IF st_config_achse.b_config_fertig THEN
	(* Fehlermeldungen und Betriebsmeldungen ab dem Startindex in die globalen Meldungsarrays schreiben *)
	garr_stoermeldungen[st_config_achse.i16_meld_startindex + 0] := st_sm.b_achse_nicht_bb;
	garr_stoermeldungen[st_config_achse.i16_meld_startindex + 1] := st_sm.b_achse_nicht_referenziert;
	garr_stoermeldungen[st_config_achse.i16_meld_startindex + 2] := st_sm.b_keine_verfahrfreigabe;
	garr_stoermeldungen[st_config_achse.i16_meld_startindex + 3] := st_sm.b_achse_nicht_auf_startpos;
	garr_stoermeldungen[st_config_achse.i16_meld_startindex + 4] := st_sm.b_ende_skalierungs_nocke;
	garr_stoermeldungen[st_config_achse.i16_meld_startindex + 5] := st_sm.b_ende_camming_nocke;
	garr_stoermeldungen[st_config_achse.i16_meld_startindex + 6] := st_sm.b_skalierung_noch_aktiv;
	garr_stoermeldungen[st_config_achse.i16_meld_startindex + 7] := FALSE;
	garr_stoermeldungen[st_config_achse.i16_meld_startindex + 8] := FALSE;
	garr_stoermeldungen[st_config_achse.i16_meld_startindex + 9] := sm_fehler_raster_oder_zaehne;
	garr_stoermeldungen[st_config_achse.i16_meld_startindex + 10] := FALSE;
	garr_stoermeldungen[st_config_achse.i16_meld_startindex + 11] := FALSE;
	garr_stoermeldungen[st_config_achse.i16_meld_startindex + 12] := sm_fehler_achse_lueften;
	garr_stoermeldungen[st_config_achse.i16_meld_startindex + 13] := sm_keine_busverbindung;
	garr_stoermeldungen[st_config_achse.i16_meld_startindex + 14] := sm_fehler_bestueckanzahl;
	garr_stoermeldungen[st_config_achse.i16_meld_startindex + 15] := sm_fehler_nach_bandwechsel;
	garr_stoermeldungen[st_config_achse.i16_meld_startindex + 16] := st_drive_cmd.meldungen.sm_write_soe_parameter;
	garr_stoermeldungen[st_config_achse.i16_meld_startindex + 17] := st_drive_cmd.meldungen.sm_read_soe_parameter;
	garr_stoermeldungen[st_config_achse.i16_meld_startindex + 18] := st_drive_cmd.meldungen.sm_write_nc_parameter;
	garr_stoermeldungen[st_config_achse.i16_meld_startindex + 19] := st_drive_cmd.meldungen.sm_read_nc_parameter;
	garr_stoermeldungen[st_config_achse.i16_meld_startindex + 20] := st_drive_cmd.meldungen.sm_power_enable;
	garr_stoermeldungen[st_config_achse.i16_meld_startindex + 21] := st_drive_cmd.meldungen.sm_power_disable;
	garr_stoermeldungen[st_config_achse.i16_meld_startindex + 22] := st_drive_cmd.meldungen.sm_reset;
	garr_stoermeldungen[st_config_achse.i16_meld_startindex + 23] := st_drive_cmd.meldungen.sm_home;
	garr_stoermeldungen[st_config_achse.i16_meld_startindex + 24] := st_drive_cmd.meldungen.sm_setposition;
	garr_stoermeldungen[st_config_achse.i16_meld_startindex + 25] := st_drive_cmd.meldungen.sm_jog_vorwaerts;
	garr_stoermeldungen[st_config_achse.i16_meld_startindex + 26] := st_drive_cmd.meldungen.sm_jog_rueckwaerts;
	garr_stoermeldungen[st_config_achse.i16_meld_startindex + 27] := st_drive_cmd.meldungen.sm_move_absolute;
	garr_stoermeldungen[st_config_achse.i16_meld_startindex + 28] := st_drive_cmd.meldungen.sm_move_relative;
	garr_stoermeldungen[st_config_achse.i16_meld_startindex + 29] := st_drive_cmd.meldungen.sm_move_velocity;
	garr_stoermeldungen[st_config_achse.i16_meld_startindex + 30] := st_drive_cmd.meldungen.sm_move_modulo;
	garr_stoermeldungen[st_config_achse.i16_meld_startindex + 31] := st_drive_cmd.meldungen.sm_stop_axis;
	garr_stoermeldungen[st_config_achse.i16_meld_startindex + 32] := st_drive_cmd.meldungen.sm_halt_axis;
	garr_stoermeldungen[st_config_achse.i16_meld_startindex + 33] := st_drive_cmd.meldungen.sm_motion_command_timeout;
	garr_stoermeldungen[st_config_achse.i16_meld_startindex + 34] := st_sm.b_achsfehler;
	garr_stoermeldungen[st_config_achse.i16_meld_startindex + 35] := st_sm.b_devicefehler;
	garr_stoermeldungen[st_config_achse.i16_meld_startindex + 36] := st_drive_cmd.meldungen.sm_limit_positiv_erreicht;
	garr_stoermeldungen[st_config_achse.i16_meld_startindex + 37] := st_drive_cmd.meldungen.sm_limit_negativ_erreicht;
	garr_stoermeldungen[st_config_achse.i16_meld_startindex + 38] := st_drive_cmd.meldungen.sm_ec_coe_sdo_write_ex;
	garr_stoermeldungen[st_config_achse.i16_meld_startindex + 39] := st_drive_cmd.meldungen.sm_ec_coe_sdo_read_ex;
	garr_stoermeldungen[st_config_achse.i16_meld_startindex + 40] := st_drive_cmd_z_achse.meldungen.sm_gear_in_slave;
	garr_stoermeldungen[st_config_achse.i16_meld_startindex + 41] := st_drive_cmd_z_achse.meldungen.sm_gear_out_slave;
	garr_stoermeldungen[st_config_achse.i16_meld_startindex + 42] := st_drive_cmd_z_achse.meldungen.sm_cam_in_slave;
	garr_stoermeldungen[st_config_achse.i16_meld_startindex + 43] := st_drive_cmd_z_achse.meldungen.sm_cam_out_slave;
	garr_stoermeldungen[st_config_achse.i16_meld_startindex + 44] := st_drive_cmd_z_achse.meldungen.sm_cam_scaleing_slave;
	garr_stoermeldungen[st_config_achse.i16_meld_startindex + 45] := st_drive_cmd_z_achse.meldungen.sm_camgear_command_timeout;
	garr_stoermeldungen[st_config_achse.i16_meld_startindex + 46] := st_drive_cmd_z_achse.meldungen.sm_read_motion_funktion_point;
	garr_stoermeldungen[st_config_achse.i16_meld_startindex + 47] := st_drive_cmd_z_achse.meldungen.sm_write_motion_funktion_point;
	garr_stoermeldungen[st_config_achse.i16_meld_startindex + 48] := st_drive_cmd_z_achse.meldungen.sm_read_camtable_slave_dynamics;
	garr_stoermeldungen[st_config_achse.i16_meld_startindex + 49] := st_drive_cmd_z_achse.meldungen.sm_read_camtable_charakteristik;
	garr_stoermeldungen[st_config_achse.i16_meld_startindex + 50] := st_drive_cmd_y_achse.meldungen.sm_gear_in_slave;
	garr_stoermeldungen[st_config_achse.i16_meld_startindex + 51] := st_drive_cmd_y_achse.meldungen.sm_gear_out_slave;
	garr_stoermeldungen[st_config_achse.i16_meld_startindex + 52] := st_drive_cmd_y_achse.meldungen.sm_cam_in_slave;
	garr_stoermeldungen[st_config_achse.i16_meld_startindex + 53] := st_drive_cmd_y_achse.meldungen.sm_cam_out_slave;
	garr_stoermeldungen[st_config_achse.i16_meld_startindex + 54] := st_drive_cmd_y_achse.meldungen.sm_cam_scaleing_slave;
	garr_stoermeldungen[st_config_achse.i16_meld_startindex + 55] := st_drive_cmd_y_achse.meldungen.sm_camgear_command_timeout;
	garr_stoermeldungen[st_config_achse.i16_meld_startindex + 56] := st_drive_cmd_y_achse.meldungen.sm_read_motion_funktion_point;
	garr_stoermeldungen[st_config_achse.i16_meld_startindex + 57] := st_drive_cmd_y_achse.meldungen.sm_write_motion_funktion_point;
	garr_stoermeldungen[st_config_achse.i16_meld_startindex + 58] := st_drive_cmd_y_achse.meldungen.sm_read_camtable_slave_dynamics;
	garr_stoermeldungen[st_config_achse.i16_meld_startindex + 59] := st_drive_cmd_y_achse.meldungen.sm_read_camtable_charakteristik;
	garr_stoermeldungen[st_config_achse.i16_meld_startindex + 60] := st_drive_cmd_b_achse.meldungen.sm_gear_in_slave;
	garr_stoermeldungen[st_config_achse.i16_meld_startindex + 61] := st_drive_cmd_b_achse.meldungen.sm_gear_out_slave;
	garr_stoermeldungen[st_config_achse.i16_meld_startindex + 62] := st_drive_cmd_b_achse.meldungen.sm_cam_in_slave;
	garr_stoermeldungen[st_config_achse.i16_meld_startindex + 63] := st_drive_cmd_b_achse.meldungen.sm_cam_out_slave;
	garr_stoermeldungen[st_config_achse.i16_meld_startindex + 64] := st_drive_cmd_b_achse.meldungen.sm_cam_scaleing_slave;
	garr_stoermeldungen[st_config_achse.i16_meld_startindex + 65] := st_drive_cmd_b_achse.meldungen.sm_camgear_command_timeout;
	garr_stoermeldungen[st_config_achse.i16_meld_startindex + 66] := st_drive_cmd_b_achse.meldungen.sm_read_motion_funktion_point;
	garr_stoermeldungen[st_config_achse.i16_meld_startindex + 67] := st_drive_cmd_b_achse.meldungen.sm_write_motion_funktion_point;
	garr_stoermeldungen[st_config_achse.i16_meld_startindex + 68] := st_drive_cmd_b_achse.meldungen.sm_read_camtable_slave_dynamics;
	garr_stoermeldungen[st_config_achse.i16_meld_startindex + 69] := st_drive_cmd_b_achse.meldungen.sm_read_camtable_charakteristik;
	garr_stoermeldungen[st_config_achse.i16_meld_startindex + 70] :=  sm_fehler_positionierung_z;
	garr_stoermeldungen[st_config_achse.i16_meld_startindex + 71] :=  sm_fehler_positionierung_y;
	garr_stoermeldungen[st_config_achse.i16_meld_startindex + 72] :=  sm_fehler_bestueckschieberanzahl;
	garr_stoermeldungen[st_config_achse.i16_meld_startindex + 73] :=  sm_fehler_bestueckposition_z;
	garr_stoermeldungen[st_config_achse.i16_meld_startindex + 74] :=  sm_fehler_bestueckposition_y;
	garr_stoermeldungen[st_config_achse.i16_meld_startindex + 75] :=  sm_fehler_positionierung_bestueckachse;
	garr_stoermeldungen[st_config_achse.i16_meld_startindex + 76] :=  st_drive_cmd_bestueckachse.meldungen.sm_gear_in_slave;
	garr_stoermeldungen[st_config_achse.i16_meld_startindex + 77] :=  st_drive_cmd_bestueckachse.meldungen.sm_gear_out_slave;
	garr_stoermeldungen[st_config_achse.i16_meld_startindex + 78] :=  st_drive_cmd_bestueckachse.meldungen.sm_cam_in_slave;
	garr_stoermeldungen[st_config_achse.i16_meld_startindex + 79] :=  st_drive_cmd_bestueckachse.meldungen.sm_cam_out_slave;
	garr_stoermeldungen[st_config_achse.i16_meld_startindex + 80] :=  st_drive_cmd_bestueckachse.meldungen.sm_camgear_command_timeout;
	garr_stoermeldungen[st_config_achse.i16_meld_startindex + 81] :=  st_drive_cmd_bestueckachse.meldungen.sm_read_motion_funktion_point;
	garr_stoermeldungen[st_config_achse.i16_meld_startindex + 82] :=  st_drive_cmd_bestueckachse.meldungen.sm_write_motion_funktion_point;
	garr_stoermeldungen[st_config_achse.i16_meld_startindex + 83] :=  st_drive_cmd_bestueckachse.meldungen.sm_read_camtable_slave_dynamics;
	garr_stoermeldungen[st_config_achse.i16_meld_startindex + 84] :=  st_drive_cmd_bestueckachse.meldungen.sm_read_camtable_charakteristik;
	garr_stoermeldungen[st_config_achse.i16_meld_startindex + 85] :=  FALSE;
	garr_stoermeldungen[st_config_achse.i16_meld_startindex + 86] :=  FALSE;
	garr_stoermeldungen[st_config_achse.i16_meld_startindex + 87] :=  FALSE;
	garr_stoermeldungen[st_config_achse.i16_meld_startindex + 88] :=  FALSE;
	garr_stoermeldungen[st_config_achse.i16_meld_startindex + 89] :=  FALSE;
	garr_stoermeldungen[st_config_achse.i16_meld_startindex + 90] :=  FALSE;
	garr_stoermeldungen[st_config_achse.i16_meld_startindex + 91] :=  FALSE;
	garr_stoermeldungen[st_config_achse.i16_meld_startindex + 92] :=  FALSE;
	garr_stoermeldungen[st_config_achse.i16_meld_startindex + 93] :=  FALSE;
	garr_stoermeldungen[st_config_achse.i16_meld_startindex + 94] :=  FALSE;
	garr_stoermeldungen[st_config_achse.i16_meld_startindex + 95] :=  FALSE;
	garr_stoermeldungen[st_config_achse.i16_meld_startindex + 96] :=  FALSE;
	garr_stoermeldungen[st_config_achse.i16_meld_startindex + 97] :=  FALSE;
	garr_stoermeldungen[st_config_achse.i16_meld_startindex + 98] :=  FALSE;
	garr_stoermeldungen[st_config_achse.i16_meld_startindex + 99] :=  FALSE;
	
	garr_betriebsmeldungen[st_config_achse.i16_meld_startindex + 0] := bm_bandende_einzug_links_erreicht;
	garr_betriebsmeldungen[st_config_achse.i16_meld_startindex + 1] := bm_einzug_links_band_entnehmen;
	garr_betriebsmeldungen[st_config_achse.i16_meld_startindex + 2] := bm_einzug_links_band_auf_anschlag;
	garr_betriebsmeldungen[st_config_achse.i16_meld_startindex + 3] := FALSE;
	garr_betriebsmeldungen[st_config_achse.i16_meld_startindex + 4] := FALSE;
	garr_betriebsmeldungen[st_config_achse.i16_meld_startindex + 5] := FALSE;
	garr_betriebsmeldungen[st_config_achse.i16_meld_startindex + 6] := FALSE;
	garr_betriebsmeldungen[st_config_achse.i16_meld_startindex + 7] := FALSE;
	garr_betriebsmeldungen[st_config_achse.i16_meld_startindex + 8] := FALSE;
	garr_betriebsmeldungen[st_config_achse.i16_meld_startindex + 9] := FALSE;
	garr_betriebsmeldungen[st_config_achse.i16_meld_startindex + 10] := bm_bandende_einzug_rechts_erreicht;
	garr_betriebsmeldungen[st_config_achse.i16_meld_startindex + 11] := bm_einzug_rechts_band_entnehmen;
	garr_betriebsmeldungen[st_config_achse.i16_meld_startindex + 12] := bm_einzug_rechts_band_auf_anschlag;
	garr_betriebsmeldungen[st_config_achse.i16_meld_startindex + 13] := FALSE;
	garr_betriebsmeldungen[st_config_achse.i16_meld_startindex + 14] := FALSE;
	garr_betriebsmeldungen[st_config_achse.i16_meld_startindex + 15] := FALSE;
	garr_betriebsmeldungen[st_config_achse.i16_meld_startindex + 16] := FALSE;
	garr_betriebsmeldungen[st_config_achse.i16_meld_startindex + 17] := FALSE;
	garr_betriebsmeldungen[st_config_achse.i16_meld_startindex + 18] := FALSE;
	garr_betriebsmeldungen[st_config_achse.i16_meld_startindex + 19] := FALSE;
	garr_betriebsmeldungen[st_config_achse.i16_meld_startindex + 20] := bm_bandende_beide_einzuege_erreicht;
	garr_betriebsmeldungen[st_config_achse.i16_meld_startindex + 21] := bm_override_kleiner_stufe9;
	garr_betriebsmeldungen[st_config_achse.i16_meld_startindex + 22] := bm_md_offset_z_pos_0_zu_hoch;
	garr_betriebsmeldungen[st_config_achse.i16_meld_startindex + 23] := bm_md_offset_y_pos_0_zu_hoch;
	garr_betriebsmeldungen[st_config_achse.i16_meld_startindex + 24] := FALSE;
	garr_betriebsmeldungen[st_config_achse.i16_meld_startindex + 25] := FALSE;
	garr_betriebsmeldungen[st_config_achse.i16_meld_startindex + 26] := FALSE;
	garr_betriebsmeldungen[st_config_achse.i16_meld_startindex + 27] := FALSE;
	garr_betriebsmeldungen[st_config_achse.i16_meld_startindex + 28] := FALSE;
	garr_betriebsmeldungen[st_config_achse.i16_meld_startindex + 29] := FALSE;
	garr_betriebsmeldungen[st_config_achse.i16_meld_startindex + 30] := FALSE;
	garr_betriebsmeldungen[st_config_achse.i16_meld_startindex + 31] := FALSE;
	garr_betriebsmeldungen[st_config_achse.i16_meld_startindex + 32] := FALSE;
	garr_betriebsmeldungen[st_config_achse.i16_meld_startindex + 33] := FALSE;
	garr_betriebsmeldungen[st_config_achse.i16_meld_startindex + 34] := FALSE;
	garr_betriebsmeldungen[st_config_achse.i16_meld_startindex + 35] := FALSE;
	garr_betriebsmeldungen[st_config_achse.i16_meld_startindex + 36] := FALSE;
	garr_betriebsmeldungen[st_config_achse.i16_meld_startindex + 37] := FALSE;
	garr_betriebsmeldungen[st_config_achse.i16_meld_startindex + 38] := FALSE;
	garr_betriebsmeldungen[st_config_achse.i16_meld_startindex + 39] := FALSE;
	garr_betriebsmeldungen[st_config_achse.i16_meld_startindex + 40] := FALSE;
	garr_betriebsmeldungen[st_config_achse.i16_meld_startindex + 41] := FALSE;
	garr_betriebsmeldungen[st_config_achse.i16_meld_startindex + 42] := FALSE;
	garr_betriebsmeldungen[st_config_achse.i16_meld_startindex + 43] := FALSE;
	garr_betriebsmeldungen[st_config_achse.i16_meld_startindex + 44] := FALSE;
	garr_betriebsmeldungen[st_config_achse.i16_meld_startindex + 45] := FALSE;
	garr_betriebsmeldungen[st_config_achse.i16_meld_startindex + 46] := FALSE;
	garr_betriebsmeldungen[st_config_achse.i16_meld_startindex + 47] := FALSE;
	garr_betriebsmeldungen[st_config_achse.i16_meld_startindex + 48] := FALSE;
	garr_betriebsmeldungen[st_config_achse.i16_meld_startindex + 49] := FALSE;
	garr_betriebsmeldungen[st_config_achse.i16_meld_startindex + 50] := FALSE;
	garr_betriebsmeldungen[st_config_achse.i16_meld_startindex + 51] := FALSE;
	garr_betriebsmeldungen[st_config_achse.i16_meld_startindex + 52] := FALSE;
	garr_betriebsmeldungen[st_config_achse.i16_meld_startindex + 53] := FALSE;
	garr_betriebsmeldungen[st_config_achse.i16_meld_startindex + 54] := FALSE;
	garr_betriebsmeldungen[st_config_achse.i16_meld_startindex + 55] := FALSE;
	garr_betriebsmeldungen[st_config_achse.i16_meld_startindex + 56] := FALSE;
	garr_betriebsmeldungen[st_config_achse.i16_meld_startindex + 57] := FALSE;
	garr_betriebsmeldungen[st_config_achse.i16_meld_startindex + 58] := FALSE;
	garr_betriebsmeldungen[st_config_achse.i16_meld_startindex + 59] := FALSE;
	garr_betriebsmeldungen[st_config_achse.i16_meld_startindex + 60] := FALSE;
	garr_betriebsmeldungen[st_config_achse.i16_meld_startindex + 61] := FALSE;
	garr_betriebsmeldungen[st_config_achse.i16_meld_startindex + 62] := FALSE;
	garr_betriebsmeldungen[st_config_achse.i16_meld_startindex + 63] := FALSE;
	garr_betriebsmeldungen[st_config_achse.i16_meld_startindex + 64] := FALSE;
	garr_betriebsmeldungen[st_config_achse.i16_meld_startindex + 65] := FALSE;
	garr_betriebsmeldungen[st_config_achse.i16_meld_startindex + 66] := FALSE;
	garr_betriebsmeldungen[st_config_achse.i16_meld_startindex + 67] := FALSE;
	garr_betriebsmeldungen[st_config_achse.i16_meld_startindex + 68] := FALSE;
	garr_betriebsmeldungen[st_config_achse.i16_meld_startindex + 69] := FALSE;
	garr_betriebsmeldungen[st_config_achse.i16_meld_startindex + 70] :=  FALSE;
	garr_betriebsmeldungen[st_config_achse.i16_meld_startindex + 71] :=  FALSE;
	garr_betriebsmeldungen[st_config_achse.i16_meld_startindex + 72] :=  FALSE;
	garr_betriebsmeldungen[st_config_achse.i16_meld_startindex + 73] :=  FALSE;
	garr_betriebsmeldungen[st_config_achse.i16_meld_startindex + 74] :=  FALSE;
	garr_betriebsmeldungen[st_config_achse.i16_meld_startindex + 75] :=  FALSE;
	garr_betriebsmeldungen[st_config_achse.i16_meld_startindex + 76] :=  FALSE;
	garr_betriebsmeldungen[st_config_achse.i16_meld_startindex + 77] :=  FALSE;
	garr_betriebsmeldungen[st_config_achse.i16_meld_startindex + 78] :=  FALSE;
	garr_betriebsmeldungen[st_config_achse.i16_meld_startindex + 79] :=  FALSE;
	garr_betriebsmeldungen[st_config_achse.i16_meld_startindex + 80] :=  FALSE;
	garr_betriebsmeldungen[st_config_achse.i16_meld_startindex + 81] :=  FALSE;
	garr_betriebsmeldungen[st_config_achse.i16_meld_startindex + 82] :=  FALSE;
	garr_betriebsmeldungen[st_config_achse.i16_meld_startindex + 83] :=  FALSE;
	garr_betriebsmeldungen[st_config_achse.i16_meld_startindex + 84] :=  FALSE;
	garr_betriebsmeldungen[st_config_achse.i16_meld_startindex + 85] :=  FALSE;
	garr_betriebsmeldungen[st_config_achse.i16_meld_startindex + 86] :=  FALSE;
	garr_betriebsmeldungen[st_config_achse.i16_meld_startindex + 87] :=  FALSE;
	garr_betriebsmeldungen[st_config_achse.i16_meld_startindex + 88] :=  FALSE;
	garr_betriebsmeldungen[st_config_achse.i16_meld_startindex + 89] :=  FALSE;
	garr_betriebsmeldungen[st_config_achse.i16_meld_startindex + 90] :=  FALSE;
	garr_betriebsmeldungen[st_config_achse.i16_meld_startindex + 91] :=  FALSE;
	garr_betriebsmeldungen[st_config_achse.i16_meld_startindex + 92] :=  FALSE;
	garr_betriebsmeldungen[st_config_achse.i16_meld_startindex + 93] :=  FALSE;
	garr_betriebsmeldungen[st_config_achse.i16_meld_startindex + 94] :=  FALSE;
	garr_betriebsmeldungen[st_config_achse.i16_meld_startindex + 95] :=  FALSE;
	garr_betriebsmeldungen[st_config_achse.i16_meld_startindex + 96] :=  FALSE;
	garr_betriebsmeldungen[st_config_achse.i16_meld_startindex + 97] :=  FALSE;
	garr_betriebsmeldungen[st_config_achse.i16_meld_startindex + 98] :=  FALSE;
	garr_betriebsmeldungen[st_config_achse.i16_meld_startindex + 99] :=  FALSE;
END_IF
END_PROGRAM
ACTION subr_ST_B_Achse:
(* Überwachung, wenn falsche Info aus dem Bestückbild kommt *)
(* Fehler, wenn mehr bestückt werden soll als das WKZ Bestückschieber hat *)
IF gst_datensatz.st_bestueckprogramm.i16_b[i16_bestueckposzaehler] > gst_datensatz.st_wkz.i16_anzahl_bestueckschieber THEN
	sm_fehler_bestueckschieberanzahl := TRUE;
	fb_state_entry.i16_next_step := FEHLER;
END_IF
END_ACTION
ACTION subr_ST_Bandeinzugsnocken_aus:
CASE gst_datensatz.st_wkz.i16_typ_bandeinzug OF
	 STANDARD_2FACH_V2:

		(* Bandeinzug: Standard_2fach_V1 *)
		gst_datensatz.st_wkz.nockenschaltwerk_bestueckachse.arr_nocken[NO_BW_BANDFAENGER_LI_EINFAHREN].b_camvalid := FALSE;
		gst_datensatz.st_wkz.nockenschaltwerk_bestueckachse.arr_nocken[NO_BW_BANDFAENGER_LI_AUSFAHREN].b_camvalid := FALSE;
		gst_datensatz.st_wkz.nockenschaltwerk_bestueckachse.arr_nocken[NO_BW_BANDKLEMMEN_LI_EINFAHREN].b_camvalid := FALSE;
		gst_datensatz.st_wkz.nockenschaltwerk_bestueckachse.arr_nocken[NO_BW_BANDKLEMMEN_LI_AUSFAHREN].b_camvalid := FALSE;
		gst_datensatz.st_wkz.nockenschaltwerk_bestueckachse.arr_nocken[NO_UW_BANDFAENGER_LI_EINFAHREN].b_camvalid := FALSE;
		gst_datensatz.st_wkz.nockenschaltwerk_bestueckachse.arr_nocken[NO_UW_BANDFAENGER_LI_AUSFAHREN].b_camvalid := FALSE;
		gst_datensatz.st_wkz.nockenschaltwerk_bestueckachse.arr_nocken[NO_UW_BANDKLEMMEN_LI_EINFAHREN].b_camvalid := FALSE;
		gst_datensatz.st_wkz.nockenschaltwerk_bestueckachse.arr_nocken[NO_UW_BANDKLEMMEN_LI_AUSFAHREN].b_camvalid := FALSE;
		gst_datensatz.st_wkz.nockenschaltwerk_bestueckachse.arr_nocken[NO_BW_BANDFAENGER_RE_EINFAHREN].b_camvalid := FALSE;
		gst_datensatz.st_wkz.nockenschaltwerk_bestueckachse.arr_nocken[NO_BW_BANDFAENGER_RE_AUSFAHREN].b_camvalid := FALSE;
		gst_datensatz.st_wkz.nockenschaltwerk_bestueckachse.arr_nocken[NO_BW_BANDKLEMMEN_RE_EINFAHREN].b_camvalid := FALSE;
		gst_datensatz.st_wkz.nockenschaltwerk_bestueckachse.arr_nocken[NO_BW_BANDKLEMMEN_RE_AUSFAHREN].b_camvalid := FALSE;
		gst_datensatz.st_wkz.nockenschaltwerk_bestueckachse.arr_nocken[NO_UW_BANDFAENGER_RE_EINFAHREN].b_camvalid := FALSE;
		gst_datensatz.st_wkz.nockenschaltwerk_bestueckachse.arr_nocken[NO_UW_BANDFAENGER_RE_AUSFAHREN].b_camvalid := FALSE;
		gst_datensatz.st_wkz.nockenschaltwerk_bestueckachse.arr_nocken[NO_UW_BANDKLEMMEN_RE_EINFAHREN].b_camvalid := FALSE;
		gst_datensatz.st_wkz.nockenschaltwerk_bestueckachse.arr_nocken[NO_UW_BANDKLEMMEN_RE_AUSFAHREN].b_camvalid := FALSE;
		(* Bandeinzug: Standard_2fach_V2 *)
		gst_datensatz.st_wkz.nockenschaltwerk_bestueckachse.arr_nocken[NO_BW_BANDFAENGER_LI_BAEZV2_EINFAHREN].b_camvalid := FALSE;
		gst_datensatz.st_wkz.nockenschaltwerk_bestueckachse.arr_nocken[NO_BW_BANDFAENGER_LI_BAEZV2_AUSFAHREN].b_camvalid := FALSE;
		gst_datensatz.st_wkz.nockenschaltwerk_bestueckachse.arr_nocken[NO_BW_BANDKLEMMEN_LI_BAEZV2_EINFAHREN].b_camvalid := FALSE;
		gst_datensatz.st_wkz.nockenschaltwerk_bestueckachse.arr_nocken[NO_BW_BANDKLEMMEN_LI_BAEZV2_AUSFAHREN].b_camvalid := FALSE;
		gst_datensatz.st_wkz.nockenschaltwerk_bestueckachse.arr_nocken[NO_BW_BANDFAENGER_RE_BAEZV2_EINFAHREN].b_camvalid := FALSE;
		gst_datensatz.st_wkz.nockenschaltwerk_bestueckachse.arr_nocken[NO_BW_BANDFAENGER_RE_BAEZV2_AUSFAHREN].b_camvalid := FALSE;
		gst_datensatz.st_wkz.nockenschaltwerk_bestueckachse.arr_nocken[NO_BW_BANDKLEMMEN_RE_BAEZV2_EINFAHREN].b_camvalid := FALSE;
		gst_datensatz.st_wkz.nockenschaltwerk_bestueckachse.arr_nocken[NO_BW_BANDKLEMMEN_RE_BAEZV2_AUSFAHREN].b_camvalid := FALSE;

		zyl_bandfaenger_li.fb.b_no_gesteuert_im_norm_betrieb := TRUE;
		zyl_bandklemmen_li.fb.b_no_gesteuert_im_norm_betrieb := TRUE;
		zyl_bandfaenger_re.fb.b_no_gesteuert_im_norm_betrieb := TRUE;
		zyl_bandklemmen_re.fb.b_no_gesteuert_im_norm_betrieb := TRUE;

	BANDWECHSLER_V2:
		(* Klemmbandeinzug ohne Sensoren *)
		gst_datensatz.st_wkz.nockenschaltwerk_bestueckachse.arr_nocken[NO_BW_BANDFAENGER_BAWEV2_EINFAHREN].b_camvalid := FALSE;
		gst_datensatz.st_wkz.nockenschaltwerk_bestueckachse.arr_nocken[NO_BW_BANDFAENGER_BAWEV2_AUSFAHREN].b_camvalid := FALSE;
		gst_datensatz.st_wkz.nockenschaltwerk_bestueckachse.arr_nocken[NO_BW_BANDKLEMMEN_BAWEV2_EINFAHREN].b_camvalid := FALSE;
		gst_datensatz.st_wkz.nockenschaltwerk_bestueckachse.arr_nocken[NO_BW_BANDKLEMMEN_BAWEV2_AUSFAHREN].b_camvalid := FALSE;

		gst_datensatz.st_wkz.nockenschaltwerk_bestueckachse.arr_nocken[NO_BW_BANDFAENGER_EINFAHREN].b_camvalid := FALSE;
		gst_datensatz.st_wkz.nockenschaltwerk_bestueckachse.arr_nocken[NO_BW_BANDFAENGER_AUSFAHREN].b_camvalid := FALSE;
		gst_datensatz.st_wkz.nockenschaltwerk_bestueckachse.arr_nocken[NO_BW_BANDKLEMMEN_EINFAHREN].b_camvalid := FALSE;
		gst_datensatz.st_wkz.nockenschaltwerk_bestueckachse.arr_nocken[NO_BW_BANDKLEMMEN_AUSFAHREN].b_camvalid := FALSE;
		gst_datensatz.st_wkz.nockenschaltwerk_bestueckachse.arr_nocken[NO_UW_BANDFAENGER_EINFAHREN].b_camvalid := FALSE;
		gst_datensatz.st_wkz.nockenschaltwerk_bestueckachse.arr_nocken[NO_UW_BANDFAENGER_AUSFAHREN].b_camvalid := FALSE;
		gst_datensatz.st_wkz.nockenschaltwerk_bestueckachse.arr_nocken[NO_UW_BANDKLEMMEN_EINFAHREN].b_camvalid := FALSE;
		gst_datensatz.st_wkz.nockenschaltwerk_bestueckachse.arr_nocken[NO_UW_BANDKLEMMEN_AUSFAHREN].b_camvalid := FALSE;

		gst_datensatz.st_wkz.nockenschaltwerk_bestueckachse.arr_nocken[NO_PNEUMATIKBANDEINZUG_GLS].b_camvalid := FALSE;
		gst_datensatz.st_wkz.nockenschaltwerk_bestueckachse.arr_nocken[NO_UW_BESTUECKSCHIEBER_ON].b_camvalid := FALSE;
		gst_datensatz.st_wkz.nockenschaltwerk_bestueckachse.arr_nocken[NO_UW_BESTUECKSCHIEBER_OFF].b_camvalid := FALSE;
		gst_datensatz.st_wkz.nockenschaltwerk_bestueckachse.arr_nocken[SP_UW_BESTUECKSCHIEBER_ON].b_camvalid := FALSE;
		gst_datensatz.st_wkz.nockenschaltwerk_bestueckachse.arr_nocken[SP_UW_BESTUECKSCHIEBER_OFF].b_camvalid := FALSE;


		zyl_bandfaenger.fb.b_no_gesteuert_im_norm_betrieb := TRUE;
		zyl_bandklemmen.fb.b_no_gesteuert_im_norm_betrieb := TRUE;

		zyl_bandfaenger.fb.b_no_gesteuert_im_norm_betrieb := TRUE;
		zyl_bandklemmen.fb.b_no_gesteuert_im_norm_betrieb := TRUE;

END_CASE;
END_ACTION
ACTION subr_ST_Bandeinzugsnocken_ein:
CASE gst_datensatz.st_wkz.i16_typ_bandeinzug OF
	 STANDARD_2FACH_V2:

		(* Bandeinzug: Standard_2fach_V2 *)
		gst_datensatz.st_wkz.nockenschaltwerk_bestueckachse.arr_nocken[NO_BW_BANDFAENGER_LI_EINFAHREN].b_camvalid := TRUE;
		gst_datensatz.st_wkz.nockenschaltwerk_bestueckachse.arr_nocken[NO_BW_BANDFAENGER_LI_AUSFAHREN].b_camvalid := TRUE;
		gst_datensatz.st_wkz.nockenschaltwerk_bestueckachse.arr_nocken[NO_BW_BANDKLEMMEN_LI_EINFAHREN].b_camvalid := TRUE;
		gst_datensatz.st_wkz.nockenschaltwerk_bestueckachse.arr_nocken[NO_BW_BANDKLEMMEN_LI_AUSFAHREN].b_camvalid := TRUE;
		gst_datensatz.st_wkz.nockenschaltwerk_bestueckachse.arr_nocken[NO_UW_BANDFAENGER_LI_EINFAHREN].b_camvalid := TRUE;
		gst_datensatz.st_wkz.nockenschaltwerk_bestueckachse.arr_nocken[NO_UW_BANDFAENGER_LI_AUSFAHREN].b_camvalid := TRUE;
		gst_datensatz.st_wkz.nockenschaltwerk_bestueckachse.arr_nocken[NO_UW_BANDKLEMMEN_LI_EINFAHREN].b_camvalid := TRUE;
		gst_datensatz.st_wkz.nockenschaltwerk_bestueckachse.arr_nocken[NO_UW_BANDKLEMMEN_LI_AUSFAHREN].b_camvalid := TRUE;
		gst_datensatz.st_wkz.nockenschaltwerk_bestueckachse.arr_nocken[NO_BW_BANDFAENGER_RE_EINFAHREN].b_camvalid := TRUE;
		gst_datensatz.st_wkz.nockenschaltwerk_bestueckachse.arr_nocken[NO_BW_BANDFAENGER_RE_AUSFAHREN].b_camvalid := TRUE;
		gst_datensatz.st_wkz.nockenschaltwerk_bestueckachse.arr_nocken[NO_BW_BANDKLEMMEN_RE_EINFAHREN].b_camvalid := TRUE;
		gst_datensatz.st_wkz.nockenschaltwerk_bestueckachse.arr_nocken[NO_BW_BANDKLEMMEN_RE_AUSFAHREN].b_camvalid := TRUE;
		gst_datensatz.st_wkz.nockenschaltwerk_bestueckachse.arr_nocken[NO_UW_BANDFAENGER_RE_EINFAHREN].b_camvalid := TRUE;
		gst_datensatz.st_wkz.nockenschaltwerk_bestueckachse.arr_nocken[NO_UW_BANDFAENGER_RE_AUSFAHREN].b_camvalid := TRUE;
		gst_datensatz.st_wkz.nockenschaltwerk_bestueckachse.arr_nocken[NO_UW_BANDKLEMMEN_RE_EINFAHREN].b_camvalid := TRUE;
		gst_datensatz.st_wkz.nockenschaltwerk_bestueckachse.arr_nocken[NO_UW_BANDKLEMMEN_RE_AUSFAHREN].b_camvalid := TRUE;
		(* Bandeinzug: Standard_2fach_V2 *)
		gst_datensatz.st_wkz.nockenschaltwerk_bestueckachse.arr_nocken[NO_BW_BANDFAENGER_LI_BAEZV2_EINFAHREN].b_camvalid := TRUE;
		gst_datensatz.st_wkz.nockenschaltwerk_bestueckachse.arr_nocken[NO_BW_BANDFAENGER_LI_BAEZV2_AUSFAHREN].b_camvalid := TRUE;
		gst_datensatz.st_wkz.nockenschaltwerk_bestueckachse.arr_nocken[NO_BW_BANDKLEMMEN_LI_BAEZV2_EINFAHREN].b_camvalid := TRUE;
		gst_datensatz.st_wkz.nockenschaltwerk_bestueckachse.arr_nocken[NO_BW_BANDKLEMMEN_LI_BAEZV2_AUSFAHREN].b_camvalid := TRUE;
		gst_datensatz.st_wkz.nockenschaltwerk_bestueckachse.arr_nocken[NO_BW_BANDFAENGER_RE_BAEZV2_EINFAHREN].b_camvalid := TRUE;
		gst_datensatz.st_wkz.nockenschaltwerk_bestueckachse.arr_nocken[NO_BW_BANDFAENGER_RE_BAEZV2_AUSFAHREN].b_camvalid := TRUE;
		gst_datensatz.st_wkz.nockenschaltwerk_bestueckachse.arr_nocken[NO_BW_BANDKLEMMEN_RE_BAEZV2_EINFAHREN].b_camvalid := TRUE;
		gst_datensatz.st_wkz.nockenschaltwerk_bestueckachse.arr_nocken[NO_BW_BANDKLEMMEN_RE_BAEZV2_AUSFAHREN].b_camvalid := TRUE;

		zyl_bandfaenger_li.fb.b_no_gesteuert_im_norm_betrieb := FALSE;
		zyl_bandklemmen_li.fb.b_no_gesteuert_im_norm_betrieb := FALSE;
		zyl_bandfaenger_re.fb.b_no_gesteuert_im_norm_betrieb := FALSE;
		zyl_bandklemmen_re.fb.b_no_gesteuert_im_norm_betrieb := FALSE;

	BANDWECHSLER_V2:
		(* Klemmbandeinzug ohne Sensoren *)
		gst_datensatz.st_wkz.nockenschaltwerk_bestueckachse.arr_nocken[NO_BW_BANDFAENGER_BAWEV2_EINFAHREN].b_camvalid := TRUE;
		gst_datensatz.st_wkz.nockenschaltwerk_bestueckachse.arr_nocken[NO_BW_BANDFAENGER_BAWEV2_AUSFAHREN].b_camvalid := TRUE;
		gst_datensatz.st_wkz.nockenschaltwerk_bestueckachse.arr_nocken[NO_BW_BANDKLEMMEN_BAWEV2_EINFAHREN].b_camvalid := TRUE;
		gst_datensatz.st_wkz.nockenschaltwerk_bestueckachse.arr_nocken[NO_BW_BANDKLEMMEN_BAWEV2_AUSFAHREN].b_camvalid := TRUE;

		gst_datensatz.st_wkz.nockenschaltwerk_bestueckachse.arr_nocken[NO_BW_BANDFAENGER_EINFAHREN].b_camvalid := TRUE;
		gst_datensatz.st_wkz.nockenschaltwerk_bestueckachse.arr_nocken[NO_BW_BANDFAENGER_AUSFAHREN].b_camvalid := TRUE;
		gst_datensatz.st_wkz.nockenschaltwerk_bestueckachse.arr_nocken[NO_BW_BANDKLEMMEN_EINFAHREN].b_camvalid := TRUE;
		gst_datensatz.st_wkz.nockenschaltwerk_bestueckachse.arr_nocken[NO_BW_BANDKLEMMEN_AUSFAHREN].b_camvalid := TRUE;
		gst_datensatz.st_wkz.nockenschaltwerk_bestueckachse.arr_nocken[NO_UW_BANDFAENGER_EINFAHREN].b_camvalid := TRUE;
		gst_datensatz.st_wkz.nockenschaltwerk_bestueckachse.arr_nocken[NO_UW_BANDFAENGER_AUSFAHREN].b_camvalid := TRUE;
		gst_datensatz.st_wkz.nockenschaltwerk_bestueckachse.arr_nocken[NO_UW_BANDKLEMMEN_EINFAHREN].b_camvalid := TRUE;
		gst_datensatz.st_wkz.nockenschaltwerk_bestueckachse.arr_nocken[NO_UW_BANDKLEMMEN_AUSFAHREN].b_camvalid := TRUE;

		gst_datensatz.st_wkz.nockenschaltwerk_bestueckachse.arr_nocken[NO_PNEUMATIKBANDEINZUG_GLS].b_camvalid := TRUE;
		gst_datensatz.st_wkz.nockenschaltwerk_bestueckachse.arr_nocken[NO_UW_BESTUECKSCHIEBER_ON].b_camvalid := b_bestueckschieber_ueberwachung_aktiv;
		gst_datensatz.st_wkz.nockenschaltwerk_bestueckachse.arr_nocken[NO_UW_BESTUECKSCHIEBER_OFF].b_camvalid := b_bestueckschieber_ueberwachung_aktiv;
		gst_datensatz.st_wkz.nockenschaltwerk_bestueckachse.arr_nocken[SP_UW_BESTUECKSCHIEBER_ON].b_camvalid := b_bestueckschieber_ueberwachung_aktiv;
		gst_datensatz.st_wkz.nockenschaltwerk_bestueckachse.arr_nocken[SP_UW_BESTUECKSCHIEBER_OFF].b_camvalid := b_bestueckschieber_ueberwachung_aktiv;

		zyl_bandfaenger.fb.b_no_gesteuert_im_norm_betrieb := TRUE;
		zyl_bandklemmen.fb.b_no_gesteuert_im_norm_betrieb := TRUE;
END_CASE;
END_ACTION
ACTION subr_ST_Bandeinzugsnocken_li_ein:
CASE gst_datensatz.st_wkz.i16_typ_bandeinzug OF
	STANDARD_2FACH_V2:

		(* Bandeinzug: Standard_2fach_V1 *)
		gst_datensatz.st_wkz.nockenschaltwerk_bestueckachse.arr_nocken[NO_BW_BANDFAENGER_LI_EINFAHREN].b_camvalid := TRUE;
		gst_datensatz.st_wkz.nockenschaltwerk_bestueckachse.arr_nocken[NO_BW_BANDFAENGER_LI_AUSFAHREN].b_camvalid := TRUE;
		gst_datensatz.st_wkz.nockenschaltwerk_bestueckachse.arr_nocken[NO_BW_BANDKLEMMEN_LI_EINFAHREN].b_camvalid := TRUE;
		gst_datensatz.st_wkz.nockenschaltwerk_bestueckachse.arr_nocken[NO_BW_BANDKLEMMEN_LI_AUSFAHREN].b_camvalid := TRUE;
		gst_datensatz.st_wkz.nockenschaltwerk_bestueckachse.arr_nocken[NO_UW_BANDFAENGER_LI_EINFAHREN].b_camvalid := TRUE;
		gst_datensatz.st_wkz.nockenschaltwerk_bestueckachse.arr_nocken[NO_UW_BANDFAENGER_LI_AUSFAHREN].b_camvalid := TRUE;
		gst_datensatz.st_wkz.nockenschaltwerk_bestueckachse.arr_nocken[NO_UW_BANDKLEMMEN_LI_EINFAHREN].b_camvalid := TRUE;
		gst_datensatz.st_wkz.nockenschaltwerk_bestueckachse.arr_nocken[NO_UW_BANDKLEMMEN_LI_AUSFAHREN].b_camvalid := TRUE;
		(* Bandeinzug: Standard_2fach_V2 *)
		gst_datensatz.st_wkz.nockenschaltwerk_bestueckachse.arr_nocken[NO_BW_BANDFAENGER_LI_BAEZV2_EINFAHREN].b_camvalid := TRUE;
		gst_datensatz.st_wkz.nockenschaltwerk_bestueckachse.arr_nocken[NO_BW_BANDFAENGER_LI_BAEZV2_AUSFAHREN].b_camvalid := TRUE;
		gst_datensatz.st_wkz.nockenschaltwerk_bestueckachse.arr_nocken[NO_BW_BANDKLEMMEN_LI_BAEZV2_EINFAHREN].b_camvalid := TRUE;
		gst_datensatz.st_wkz.nockenschaltwerk_bestueckachse.arr_nocken[NO_BW_BANDKLEMMEN_LI_BAEZV2_AUSFAHREN].b_camvalid := TRUE;

		zyl_bandfaenger_li.fb.b_no_gesteuert_im_norm_betrieb := FALSE;
		zyl_bandklemmen_li.fb.b_no_gesteuert_im_norm_betrieb := FALSE;
		zyl_bandfaenger_re.fb.b_no_gesteuert_im_norm_betrieb := FALSE;
		zyl_bandklemmen_re.fb.b_no_gesteuert_im_norm_betrieb := FALSE;

END_CASE;
END_ACTION
ACTION subr_ST_Bandeinzugsnocken_re_ein:
CASE gst_datensatz.st_wkz.i16_typ_bandeinzug OF
	STANDARD_2FACH_V2:

		(* Bandeinzug: Standard_2fach_V1 *)
		gst_datensatz.st_wkz.nockenschaltwerk_bestueckachse.arr_nocken[NO_BW_BANDFAENGER_RE_EINFAHREN].b_camvalid := TRUE;
		gst_datensatz.st_wkz.nockenschaltwerk_bestueckachse.arr_nocken[NO_BW_BANDFAENGER_RE_AUSFAHREN].b_camvalid := TRUE;
		gst_datensatz.st_wkz.nockenschaltwerk_bestueckachse.arr_nocken[NO_BW_BANDKLEMMEN_RE_EINFAHREN].b_camvalid := TRUE;
		gst_datensatz.st_wkz.nockenschaltwerk_bestueckachse.arr_nocken[NO_BW_BANDKLEMMEN_RE_AUSFAHREN].b_camvalid := TRUE;
		gst_datensatz.st_wkz.nockenschaltwerk_bestueckachse.arr_nocken[NO_UW_BANDFAENGER_RE_EINFAHREN].b_camvalid := TRUE;
		gst_datensatz.st_wkz.nockenschaltwerk_bestueckachse.arr_nocken[NO_UW_BANDFAENGER_RE_AUSFAHREN].b_camvalid := TRUE;
		gst_datensatz.st_wkz.nockenschaltwerk_bestueckachse.arr_nocken[NO_UW_BANDKLEMMEN_RE_EINFAHREN].b_camvalid := TRUE;
		gst_datensatz.st_wkz.nockenschaltwerk_bestueckachse.arr_nocken[NO_UW_BANDKLEMMEN_RE_AUSFAHREN].b_camvalid := TRUE;
		(* Bandeinzug: Standard_2fach_V2 *)
		gst_datensatz.st_wkz.nockenschaltwerk_bestueckachse.arr_nocken[NO_BW_BANDFAENGER_RE_BAEZV2_EINFAHREN].b_camvalid := TRUE;
		gst_datensatz.st_wkz.nockenschaltwerk_bestueckachse.arr_nocken[NO_BW_BANDFAENGER_RE_BAEZV2_AUSFAHREN].b_camvalid := TRUE;
		gst_datensatz.st_wkz.nockenschaltwerk_bestueckachse.arr_nocken[NO_BW_BANDKLEMMEN_RE_BAEZV2_EINFAHREN].b_camvalid := TRUE;
		gst_datensatz.st_wkz.nockenschaltwerk_bestueckachse.arr_nocken[NO_BW_BANDKLEMMEN_RE_BAEZV2_AUSFAHREN].b_camvalid := TRUE;
		
		zyl_bandfaenger_li.fb.b_no_gesteuert_im_norm_betrieb := FALSE;
		zyl_bandklemmen_li.fb.b_no_gesteuert_im_norm_betrieb := FALSE;
		zyl_bandfaenger_re.fb.b_no_gesteuert_im_norm_betrieb := FALSE;
		zyl_bandklemmen_re.fb.b_no_gesteuert_im_norm_betrieb := FALSE;

END_CASE;
END_ACTION
ACTION subr_ST_Cam_B_Achse:
(* B-Achse *)
fb_axis_b_achse.st_camscaling_data.SlaveScaling :=
	F_Servobandeinzug_Strecke_zu_Grad(
		strecke := INT_TO_LREAL(gst_datensatz.st_bestueckprogramm.i16_b[i16_bestueckposzaehler])
			* gst_datensatz.st_band.r_raster);

IF b_achse.Status.CamScalingPending THEN
	st_sm.b_skalierung_noch_aktiv := TRUE;
	fb_state_entry.i16_next_step := FEHLER;
ELSE
	IF b_achse.NcToPlc.CoupleState = 0 THEN
		st_drive_cmd_b_achse.enu_cmd := CAM_IN_SLAVE;
	ELSE
		st_drive_cmd_b_achse.enu_cmd := CAM_SCALEING_SLAVE;
	END_IF
END_IF
END_ACTION
ACTION subr_ST_Cam_Bestueck_Maschine:
CASE gst_datensatz.st_md.i16_typ_zelle OF
	KEINE_ZELLE:
		;
	BESTUECKZELLE_1700, BESTUECKZELLE_1720:
		subr_ST_Cam_Bestueckachse();

	RASTERFOLIE:
		;
END_CASE
END_ACTION
ACTION subr_ST_Cam_Bestueckachse:
(* Bestueckachse *)
IF gst_datensatz.st_bestueckprogramm.i16_b[i16_bestueckposzaehler] <= 0 THEN
	i16_bestueckachse_cam_table_id := 6;	(* 0-Scalierung *)
	subr_ST_Bandeinzugsnocken_aus();
ELSE
	i16_bestueckachse_cam_table_id := 5;	(* 1-Scalierung *)
	subr_ST_Bandeinzugsnocken_ein();
END_IF

IF i16_bestueckachse_cam_table_id <> i16_bestueckachse_cam_table_id_alt THEN
	fb_axis_bestueckachse.mc_activation_mode_camin:= MC_CAMACTIVATION_ATMASTERCAMPOS;
	fb_axis_bestueckachse.lr_activation_position_camin := gst_datensatz.st_md.st_md_bestueckachse.lr_startposition;
	st_drive_cmd_bestueckachse.enu_cmd := CAM_IN_SLAVE;
	i16_bestueckachse_cam_table_id_alt := i16_bestueckachse_cam_table_id;
END_IF
END_ACTION
ACTION subr_ST_Cam_Y_Achse:
(* Y-Achse *)
IF i16_bestueckposzaehler = 0 THEN
	lr_ErsteBestueckposY := gst_datensatz.st_isk.lr_pos_y_0 +
						gst_datensatz.st_wkz.lr_offset_y_pos_0 +
						gst_datensatz.st_wt.lr_offset_y_pos_0 +
						gst_datensatz.st_md.lr_offset_y_pos_0 +
						gst_datensatz.st_bestueckprogramm.lr_y[0];
	fb_axis_y_achse.st_camscaling_data.SlaveScaling := fb_berechnung_override_achse.lr_skalierung_slave_achse2 := lr_ErsteBestueckposY - y_achse.NcToPlc.ActPos;
	(* Falls die Positionierung Probleme macht, könnte man auch so rechnen *)
	(*fb_axis_y_achse.st_camscaling_data.SlaveScaling := fb_berechnung_override_achse.lr_skalierung_slave_achse2 := lr_ErsteBestueckposY - gst_datensatz.st_wkz.r_wkz_einfahrpos_y;*)
ELSIF i16_bestueckposzaehler > 0 AND i16_bestueckposzaehler < gst_datensatz.st_bestueckprogramm.i32_anzahl THEN
	fb_axis_y_achse.st_camscaling_data.SlaveScaling := fb_berechnung_override_achse.lr_skalierung_slave_achse2 := gst_datensatz.st_bestueckprogramm.lr_y[i16_bestueckposzaehler] - gst_datensatz.st_bestueckprogramm.lr_y[i16_bestueckposzaehler - 1];
ELSE
	fb_axis_y_achse.st_camscaling_data.SlaveScaling := fb_berechnung_override_achse.lr_skalierung_slave_achse2 := 0.0;
END_IF
IF y_achse.Status.CamScalingPending THEN
	st_sm.b_skalierung_noch_aktiv := TRUE;
	fb_state_entry.i16_next_step := FEHLER;
ELSE
	IF y_achse.NcToPlc.CoupleState = 0 THEN
		st_drive_cmd_y_achse.enu_cmd := CAM_IN_SLAVE;
	ELSE
		st_drive_cmd_y_achse.enu_cmd := CAM_SCALEING_SLAVE;
	END_IF
END_IF
END_ACTION
ACTION subr_ST_Cam_Z_Achse:
(* Z-Achse *)
IF i16_bestueckposzaehler > 0 AND i16_bestueckposzaehler < gst_datensatz.st_bestueckprogramm.i32_anzahl THEN
	fb_axis_z_achse.st_camscaling_data.SlaveScaling := fb_berechnung_override_achse.lr_skalierung_slave_achse1 := gst_datensatz.st_bestueckprogramm.lr_z[i16_bestueckposzaehler] - gst_datensatz.st_bestueckprogramm.lr_z[i16_bestueckposzaehler - 1];
ELSE
	fb_axis_z_achse.st_camscaling_data.SlaveScaling := fb_berechnung_override_achse.lr_skalierung_slave_achse1 := 0.0;
END_IF
IF z_achse.Status.CamScalingPending THEN
	st_sm.b_skalierung_noch_aktiv := TRUE;
	fb_state_entry.i16_next_step := FEHLER;
ELSE
	IF z_achse.NcToPlc.CoupleState = 0 THEN
		st_drive_cmd_z_achse.enu_cmd := CAM_IN_SLAVE;
	ELSE
		st_drive_cmd_z_achse.enu_cmd := CAM_SCALEING_SLAVE;
	END_IF
END_IF
END_ACTION
ACTION subr_ST_EinzugLueften:
(* SP_SERVOBANDEINZUG_LUEFTEN niemals vorsteuern *)
gst_datensatz.st_wkz.nockenschaltwerk_bestueckachse.arr_nocken[SP_SERVOBANDEINZUG_LUEFTEN].t_vorsteuerzeit := t#0ms;

fb_r_trig_bandeinzug_lueften(CLK:= nockenschaltwerk_bestueckachse.fb.arr_spur[SP_SERVOBANDEINZUG_LUEFTEN], Q=> );
fb_f_trig_bandeinzug_lueften(CLK:= nockenschaltwerk_bestueckachse.fb.arr_spur[SP_SERVOBANDEINZUG_LUEFTEN], Q=> );

(* Abschalten, falls die Schrittkette beim Lüften aus irgendwelchen Gründen hängen bleibt *)
IF fb_r_trig_bandeinzug_lueften.Q AND
	i16_step_lueften > 0 THEN
		sm_fehler_achse_lueften := TRUE;
		fb_state_entry.i16_next_step := FEHLER;
END_IF


(* Schrittkette zum Einzug in Regelung setzen mit Positionsangleich  *)
CASE i16_step_lueften OF
(*=======================================================*)
	0:	(* CAM Out bei R Trig Lueftnocke *)

		(*-----------------------Weiterschaltbedingungen----------------------------*)
		IF fb_r_trig_bandeinzug_lueften.Q AND
			bestueckachse.NcToPlc.CoupleState <> 0 AND
			((NOT b_einfaedeln_aktiv_servo AND
			(* Bei einer Umfahrung soll Servo nicht lüften, weil die Fänger des WKZ das Band nicht halten *)
			gst_datensatz.st_bestueckprogramm.i16_b[i16_bestueckposzaehler] >= 1 ) OR
			(b_einfaedeln_aktiv_servo AND
			i16_einfaedelzaehler >= gst_datensatz.st_wkz.i16_einfaedelhub_lueften)) THEN		(* Nach x Einfädelhüben ist Band sicher im WKZ, dann darf Servobaneinzug wieder entlüften *)
			st_drive_cmd_b_achse.enu_cmd := CAM_OUT_SLAVE;
			i16_step_lueften := 10;
		END_IF

(*=======================================================*)
	10:

		(*-----------------------Weiterschaltbedingungen----------------------------*)
		IF st_drive_cmd_b_achse.enu_cmd = NO_COMMAND THEN
			ST_Servobandeinzug.i_Stromlimit := ST_Servobandeinzug.i16_lueft_torque;
			i16_step_lueften := 20;
		END_IF

(*=======================================================*)
	20: (* HOME Servobandeinzug bei F Trig Lueftnocke *)

		(*-----------------------Weiterschaltbedingungen----------------------------*)
		IF fb_f_trig_bandeinzug_lueften.Q THEN
			axis_bandeinzug_achse.st_ctrl.in.b_home := TRUE;
			i16_step_lueften := 30;
		END_IF

(*=======================================================*)
	30:

		(*-----------------------Weiterschaltbedingungen----------------------------*)
		IF axis_bandeinzug_achse.st_ctrl.out.b_fertig_2 THEN
			axis_bandeinzug_achse.st_ctrl.in.b_home := FALSE;
			i16_step_lueften := 0;
		END_IF

END_CASE
END_ACTION
ACTION subr_ST_PosUW_Bestueckachse:
(* Wenn die Betückachse von der Virtuellen Achse entkoppelt wird, muss dauerhaft der OT Sensor belegt sein.
Überwachung, ob das Auskoppeln rechtzeitig gemacht wird. Ab 300 Hub gibt es Probleme *)
IF i16_bestueckachse_cam_table_id = 6 AND NOT ST_Bestueckachse.e_referenz_sensor THEN
	sm_fehler_positionierung_bestueckachse := TRUE;
	fb_state_entry.i16_next_step := FEHLER;
END_IF
END_ACTION
ACTION subr_ST_PosUW_YZ_Achse:
(* Y *)
(* Kontrolle der Skalierungsposition der Achse nach dem Setzen eines Pins *)
IF ABS(y_achse.NcToPlc.ActPos - (lr_merker_y_pos + gst_datensatz.st_bestueckprogramm.lr_y[i16_bestueckposzaehler])) > 0.1THEN
	sm_fehler_bestueckposition_y := TRUE;
	fb_state_entry.i16_next_step := FEHLER;
END_IF

(* Überwachung auf Kommando abgeschlossen. Zusätzliche Kontrolle auf Ausführung des Skalierungskommandos *)
IF st_drive_cmd_y_achse.enu_cmd <> NO_COMMAND THEN
	st_sm.b_ende_camming_nocke := TRUE;
	fb_state_entry.i16_next_step := FEHLER;
END_IF

(* Z *)
(* Kontrolle der Skalierungsposition der Achse nach dem Setzen eines Pins *)
IF ABS(z_achse.NcToPlc.ActPos - (lr_merker_z_pos + gst_datensatz.st_bestueckprogramm.lr_z[i16_bestueckposzaehler])) > 0.2THEN
	sm_fehler_bestueckposition_z := TRUE;
	fb_state_entry.i16_next_step := FEHLER;
END_IF

(* Überwachung auf Kommando abgeschlossen. Zusätzliche Kontrolle auf Ausführung des Skalierungskommandos *)
IF st_drive_cmd_z_achse.enu_cmd <> NO_COMMAND THEN
	st_sm.b_ende_camming_nocke := TRUE;
	fb_state_entry.i16_next_step := FEHLER;
END_IF

(* Pythagoras YZ *)
(*	tv + gg: 10.08.2021
	Wir müssen nicht nur jede Achse einzeln überwachen, sondern beide Achsen zusammen überwachen.
	Bsp. 74pol 2-Fach WT: Es gibt hier Sprünge die nur 0.04 in Y Verschoben, welche dann die 
	Überwachung in Y-Achse ausgelöst hat, obwohl alles funktionert hat. Z Pos ist um 5 mm verschoben*)

(* Kontrolle, ob die Achsen gegenüber dem letzten Bestückhub weiter gefahren ist *)
lr_merker_y_pos_neu := y_achse.NcToPlc.ActPos;
lr_merker_z_pos_neu := z_achse.NcToPlc.ActPos;

lr_abstand_yz := SQRT(	EXPT(lr_merker_y_pos_alt - lr_merker_y_pos_neu, 2) +
						EXPT(lr_merker_z_pos_alt - lr_merker_z_pos_neu, 2));

IF 	(fb_axis_y_achse.st_camscaling_data.SlaveScaling <> 0 OR
	fb_axis_z_achse.st_camscaling_data.SlaveScaling <> 0) AND
	lr_abstand_yz < 0.05
THEN
	sm_fehler_positionierung_y := TRUE;
	sm_fehler_positionierung_z := TRUE;
	fb_state_entry.i16_next_step := FEHLER;
END_IF

lr_merker_y_pos_alt := lr_merker_y_pos_neu;
lr_merker_z_pos_alt := lr_merker_z_pos_neu;
END_ACTION
ACTION subr_ST_PosUW_Z_Achse:
(* Kontrolle der Skalierungsposition der Achse nach dem Setzen eines Pins *)
IF ABS(z_achse.NcToPlc.ActPos - (lr_merker_z_pos + gst_datensatz.st_bestueckprogramm.lr_z[i16_bestueckposzaehler])) > 0.2THEN
	sm_fehler_bestueckposition_z := TRUE;
	fb_state_entry.i16_next_step := FEHLER;
END_IF

(* Überwachung auf Kommando abgeschlossen. Zusätzliche Kontrolle auf Ausführung des Skalierungskommandos *)
IF st_drive_cmd_z_achse.enu_cmd <> NO_COMMAND THEN
	st_sm.b_ende_camming_nocke := TRUE;
	fb_state_entry.i16_next_step := FEHLER;
END_IF

(* Kontrolle, ob die Achse gegenüber dem letzten Bestückhub weiter gefahren ist *)
lr_merker_z_pos_neu := z_achse.NcToPlc.ActPos;
IF fb_axis_z_achse.st_camscaling_data.SlaveScaling <> 0 THEN
	IF ABS(lr_merker_z_pos_alt - lr_merker_z_pos_neu) > 0.05 THEN
		lr_merker_z_pos_alt := lr_merker_z_pos_neu;
	ELSE
		sm_fehler_positionierung_z := TRUE;
		fb_state_entry.i16_next_step := FEHLER;
	END_IF
END_IF
END_ACTION

(* POU EPT Lib/Achsen/BECKHOFF/ST_AxisJobCtrl_Motion, ST *)
FUNCTION_BLOCK ST_AxisJobCtrl_Motion
VAR_INPUT
	e_referenznocken						: BOOL;
	b_refsensor_vorhanden				: BOOL;
	b_limitsensor_positiv_vorhanden		: BOOL;
	b_limitsensor_negativ_vorhanden		: BOOL;
	i16_achstyp							: enum_ecd_typ;
	lr_override_vorgabe					: LREAL;
	st_position							: struct_ecd_positionen;
	mc_richtung_modulo					: MC_Direction;
	mc_richtung_velocity					: MC_Direction;
											(*default: MC_Positive_Direction := 1,
											MC_Shortest_Way ,
									    		MC_Negative_Direction,
									    		MC_Current_Direction *)
	mc_referenzmodus 					: MC_HomingMode; (* default: MC_DefaultHoming   default homing as defined in the SystemManager encoder parameters *)
	mc_buffermode_axis					: MC_BufferMode;     (*	MC_Aborting,	->sofortiger Abbruch der momentanen Bewegung, bei einem neuen Verfahrbefehl
														MC_Buffered,
														MC_BlendingLow,
														MC_BlendingPrevious,
														MC_BlendingNext,
														MC_BlendingHigh *)
	ui16_soeparam_write_value				: UINT;
	w_idn								: WORD;
	i16_nc_parameter_nummer				: INT;
	r_wert_nc_write_parameter				: LREAL;
	st_vorgabe_geschwindigkeiten			: struct_ecd_geschwindigkeiten;
	lr_soll_geschwindigkeit					: LREAL;
	b_bedingung_sls						: BOOL;
	st_ads_info							: struct_ads_info;
	st_eccoe_sdo						: struct_eccoe_sdo;
	b_TriggerInput						: BOOL;
	b_FallingEdge						: BOOL;
END_VAR
VAR_OUTPUT
	ui16_soeparam_read_value			: UINT;
	r_wert_nc_read_parameter				: LREAL;
	lr_RecPos							: LREAL;
END_VAR
VAR_IN_OUT
	st_masterachse						: AXIS_REF;
	st_visu_axis							: struct_ecd_visu;
	st_ecd_cmd							: struct_ecd_cmd;
END_VAR
VAR
	fb_ton_cmd_timeout					: TON;
	t_cmd_timeout						: TIME;
	t_ads_timeout							: TIME;
	fb_ton_vz							: TON;
	b_jog_vorwaerts_execute				: BOOL := FALSE;
	b_jog_rueckwaerts_execute				: BOOL := FALSE;
	e_limit_sensor_positive				AT %I* : BOOL;
	e_limit_sensor_negative				AT %I* : BOOL;
	e_referenz_sensor						AT %I* : BOOL;
	fb_f_trig_limit_sensor_positiv			: F_TRIG;
	fb_f_trig_limit_sensor_negativ			: F_TRIG;
	fb_cmd_history						: ST_CommandHistory;

	mc_power_axis 						: MC_Power;
	mc_reset_axis						: MC_Reset;
	mc_home_axis 						: MC_Home;
	mc_setposition_axis					: MC_SetPosition;
	mc_jog_axis							: MC_Jog;
	mc_moveabsolute_axis 				: MC_MoveAbsolute;
	mc_moveabsolutenext_axis 			: MC_MoveAbsolute;
	mc_moverelative_axis 					: MC_MoveRelative;
	mc_movevelocity_axis 					: MC_MoveVelocity;
	mc_movemodulo_axis					: MC_MoveModulo;
	mc_stop_axis 						: MC_Stop;
	mc_halt_axis							: MC_Halt;
	mc_touch_probe					: MC_TouchProbe;
	mc_abort_trigger						: MC_AbortTrigger;
	TriggerInput							:TRIGGER_REF;
	err_id								: DWORD := 0;
	fb_state_entry							: ST_StateEntry;
	fb_soe_reset							: FB_SoEReset;
	fb_soe_write							: FB_SoEWrite;
	fb_soe_read							: FB_SoERead;
	fb_ec_coe_sdo_write_ex				: FB_EcCoESdoWriteEx;
	fb_ec_coe_sdo_read_ex				: FB_EcCoESdoReadEx;
	mc_write_nc_parameter				: MC_WriteParameter;
	mc_read_nc_parameter				: MC_ReadParameter;
	fb_ads_write							: ADSWRITE;
	fb_ads_read							: ADSREAD;
	lr_override							: LREAL := 0.0;
	lr_override_reduziert					: LREAL := 0.0;
	lr_reduktionsfaktor						: LREAL := 5.0;
	lr_hm_master_act_velo					: LREAL := 0.0;
	lr_sollgeschwindigkeit					: LREAL := 0.0;
END_VAR
sub_TouchProbe();
(* Zeiten *)
fb_ton_cmd_timeout(IN:= , PT:=t_cmd_timeout, Q=> , ET=> );
fb_ton_vz(IN:= , PT:= , Q=> , ET=> );

(* Flanken *)
fb_f_trig_limit_sensor_positiv(CLK:= e_limit_sensor_positive, Q=> );
fb_f_trig_limit_sensor_negativ(CLK:= e_limit_sensor_negative, Q=> );

(* =====Beschränkung des Overrides wegen SLS bei offenen Türen===== *)
IF b_bedingung_sls THEN
	IF i16_achstyp = RUND OR  i16_achstyp = RUND_VIRTUELL THEN
		lr_hm_master_act_velo := st_masterachse.NcToPlc.ActVelo * 60 / 360;
	ELSE
		lr_hm_master_act_velo := st_masterachse.NcToPlc.ActVelo;
	END_IF
	IF ABS(lr_hm_master_act_velo) < st_vorgabe_geschwindigkeiten.lr_jog THEN
		lr_override := lr_override_reduziert := lr_override_vorgabe;
	ELSE
		lr_override_reduziert := lr_override_reduziert - lr_reduktionsfaktor;
		IF lr_override_reduziert >= 0 OR lr_override_reduziert <= 100 THEN
			lr_override := lr_override_reduziert;
		END_IF
	END_IF
ELSE
	lr_override := lr_override_vorgabe;
END_IF

(* =====Beschränkung der Achsgeschwindigkeiten===== *)
(* Verrechnet nach Rund/Linear wird weiter unten *)
lr_sollgeschwindigkeit := lr_soll_geschwindigkeit;

(* Beschränkung der Geschwindigkeit *)
IF lr_sollgeschwindigkeit > st_vorgabe_geschwindigkeiten.lr_auto_max THEN
	lr_sollgeschwindigkeit := st_vorgabe_geschwindigkeiten.lr_auto_max;
ELSIF lr_sollgeschwindigkeit < st_vorgabe_geschwindigkeiten.lr_auto_min THEN
	lr_sollgeschwindigkeit := st_vorgabe_geschwindigkeiten.lr_auto_min ;
END_IF

(* ======Ausgabe von Position und Geschwindigkeit der Achse===== *)
IF i16_achstyp = RUND OR  i16_achstyp = RUND_VIRTUELL THEN
	(* INT-Daten *)
	IF LREAL_TO_DINT(st_masterachse.NcToPlc.ModuloActPos) = 360 THEN
		st_visu_axis.i32_position_ist := 0;
	ELSE
		st_visu_axis.i32_position_ist := LREAL_TO_DINT(st_masterachse.NcToPlc.ModuloActPos);
	END_IF
	st_visu_axis.i32_geschwindigkeit_ist := LREAL_TO_DINT(st_masterachse.NcToPlc.ActVelo * 60 / 360); (* Hub = Grad/sec / 360 * 60s *)

	(* LREAL-DATEN *)
	st_visu_axis.lr_position_ist :=st_masterachse.NcToPlc.ModuloActPos;
	st_visu_axis.lr_geschwindigkeit_ist := st_masterachse.NcToPlc.ActVelo * 60 / 360; (* Hub = Grad/sec / 360 * 60s *)
ELSIF i16_achstyp = LINEAR OR i16_achstyp = LINEAR_VIRTUELL THEN
	st_visu_axis.lr_position_ist :=st_masterachse.NcToPlc.ActPos;
	st_visu_axis.lr_geschwindigkeit_ist := st_masterachse.NcToPlc.ActVelo;
ELSE
	st_visu_axis.lr_position_ist :=st_masterachse.NcToPlc.ActPos;
	st_visu_axis.lr_geschwindigkeit_ist := st_masterachse.NcToPlc.ActVelo;
END_IF

(* ======================================Schrittkette Drivebefehle======================================== *)
fb_state_entry(
	i16_next_step:= , 
	i16_pos:= 1,
	s_debugtext:= ,
	E=> ,
	X=> ,
	i16_step=> ,
	i16_last_step=> );

CASE fb_state_entry.i16_step OF
(*=======================================================*)
	0:	(* Init *)
		st_ecd_cmd.b_job_fehler := FALSE;
		st_ecd_cmd.enu_cmd := NO_COMMAND;
		mc_buffermode_axis := MC_Aborting;
		t_cmd_timeout := T#10s;
		t_ads_timeout := t#10s;
		err_id :=0;

		b_jog_vorwaerts_execute := FALSE;
		b_jog_rueckwaerts_execute := FALSE;
		mc_power_axis.Enable := FALSE;
		mc_reset_axis.Execute := FALSE;
		mc_home_axis.Execute := FALSE;
		mc_moveabsolute_axis.Execute := FALSE;
		mc_moverelative_axis.Execute := FALSE;
		mc_movevelocity_axis.Execute := FALSE;
		mc_movemodulo_axis.Execute := FALSE;
		mc_setposition_axis.Execute := FALSE;
		mc_halt_axis.Execute := FALSE;
		mc_stop_axis.Execute := FALSE;
		mc_touch_probe.Execute := FALSE;
		fb_soe_reset.Execute := FALSE;
		fb_soe_write.Execute := FALSE;
		fb_soe_read.Execute := FALSE;
		fb_ec_coe_sdo_write_ex.bExecute := FALSE;
		fb_ec_coe_sdo_write_ex.bExecute := FALSE;
		mc_write_nc_parameter.Execute := FALSE;
		mc_read_nc_parameter.Enable := FALSE;
		fb_ads_write.WRITE := FALSE;
		fb_ads_read.READ := FALSE;

		st_ecd_cmd.meldungen.sm_power_enable := FALSE;
		st_ecd_cmd.meldungen.sm_power_disable := FALSE;
		st_ecd_cmd.meldungen.sm_reset := FALSE;
		st_ecd_cmd.meldungen.sm_home := FALSE;
		st_ecd_cmd.meldungen.sm_setposition := FALSE;
		st_ecd_cmd.meldungen.sm_jog_vorwaerts := FALSE;
		st_ecd_cmd.meldungen.sm_jog_rueckwaerts := FALSE;
		st_ecd_cmd.meldungen.sm_move_absolute := FALSE;
		st_ecd_cmd.meldungen.sm_move_relative := FALSE;
		st_ecd_cmd.meldungen.sm_move_velocity := FALSE;
		st_ecd_cmd.meldungen.sm_move_modulo := FALSE;
		st_ecd_cmd.meldungen.sm_stop_axis := FALSE;
		st_ecd_cmd.meldungen.sm_halt_axis := FALSE;
		st_ecd_cmd.meldungen.sm_motion_command_timeout := FALSE;
		st_ecd_cmd.meldungen.sm_limit_positiv_erreicht := FALSE;
		st_ecd_cmd.meldungen.sm_limit_negativ_erreicht := FALSE;
		st_ecd_cmd.meldungen.sm_write_soe_parameter := FALSE;
		st_ecd_cmd.meldungen.sm_read_soe_parameter := FALSE;
		st_ecd_cmd.meldungen.sm_write_nc_parameter := FALSE;
		st_ecd_cmd.meldungen.sm_read_nc_parameter := FALSE;
		st_ecd_cmd.meldungen.sm_write_ads_parameter := FALSE;
		st_ecd_cmd.meldungen.sm_read_ads_parameter := FALSE;
		st_ecd_cmd.meldungen.sm_ec_coe_sdo_write_ex := FALSE;
		st_ecd_cmd.meldungen.sm_ec_coe_sdo_read_ex := FALSE;
		st_ecd_cmd.meldungen.sm_touch_probe_defect := FALSE;
		st_ecd_cmd.meldungen.sm_touch_probe_err := FALSE;
		fb_state_entry.i16_next_step := 1;

(*=======================================================*)
	1:	(* Warte auf Kommando *)
		IF st_ecd_cmd.enu_cmd > NO_COMMAND THEN
			IF st_ecd_cmd.enu_cmd <= HALT_AXIS THEN
				(* Wichtige Kommandos werden mit Direktsprung ausgeführt, um Zykluszeit zu sparen *)
				IF st_ecd_cmd.enu_cmd = HALT_AXIS THEN
					fb_state_entry.i16_next_step := 120;
				ELSIF st_ecd_cmd.enu_cmd = STOP_AXIS THEN
					fb_state_entry.i16_next_step := 130;
				ELSE
					fb_state_entry.i16_next_step := 10;	(* Motionbefehle *)
				END_IF
			ELSE
				fb_state_entry.i16_next_step := 500;	(* Parameter für Achsen *)
			END_IF
		END_IF

(*=======================Motionbefehle================================*)
	10:	(* Power OFF NC-Achse *)
		fb_ton_cmd_timeout.IN := TRUE;
		IF st_ecd_cmd.enu_cmd = POWER_DISABLE THEN
			mc_power_axis.Enable := FALSE;
			fb_state_entry.i16_next_step := 11;
		ELSE
			fb_ton_cmd_timeout.IN := FALSE;
			fb_state_entry.i16_next_step := 20;
		END_IF
	11:
		CASE i16_achstyp OF
			LINEAR, RUND:
				IF NOT mc_power_axis.Status AND NOT st_masterachse.Status.Operational THEN
					fb_state_entry.i16_next_step := 999;
				ELSIF NOT mc_power_axis.Busy AND mc_power_axis.Error THEN
					err_id := mc_power_axis.ErrorID;
					st_ecd_cmd.meldungen.sm_power_disable := TRUE;
					fb_state_entry.i16_next_step := 1000;
				END_IF
			LINEAR_VIRTUELL, RUND_VIRTUELL:
				IF NOT mc_power_axis.Busy AND mc_power_axis.Error THEN
					err_id := mc_power_axis.ErrorID;
					st_ecd_cmd.meldungen.sm_power_disable := TRUE;
					fb_state_entry.i16_next_step := 1000;
				ELSE
					fb_state_entry.i16_next_step := 999;
				END_IF
			SERVOKLEMME7201:
				IF NOT mc_power_axis.Status AND NOT st_masterachse.Status.Operational THEN
					fb_state_entry.i16_next_step := 999;
				ELSIF NOT mc_power_axis.Busy AND mc_power_axis.Error THEN
					err_id := mc_power_axis.ErrorID;
					st_ecd_cmd.meldungen.sm_power_disable := TRUE;
					fb_state_entry.i16_next_step := 1000;
				END_IF
		END_CASE

(*=======================================================*)
	20:	(* Reset NC-Achse und Servokontroller*)
		IF	st_ecd_cmd.enu_cmd = RESET OR
			st_masterachse.Status.DriveDeviceError OR
			st_masterachse.Status.Error
			 THEN
			fb_state_entry.i16_next_step := 21;
		ELSE
			fb_state_entry.i16_next_step := 30;
		END_IF
	21:	(*  Reset AX5000 Fehler  *)
		CASE i16_achstyp OF
			LINEAR, RUND:
				IF NOT st_masterachse.Status.DriveDeviceError THEN
					fb_state_entry.i16_next_step := 24;
				ELSE
					fb_ton_cmd_timeout.IN := TRUE;
					fb_soe_reset.Execute := TRUE;
					IF fb_soe_reset.Busy THEN
						fb_state_entry.i16_next_step := 22;
					END_IF
				END_IF
			LINEAR_VIRTUELL, RUND_VIRTUELL, SERVOKLEMME7201:
				fb_state_entry.i16_next_step := 24;
		END_CASE
	22:
		IF NOT fb_soe_reset.Busy THEN
			IF  fb_soe_reset.Error THEN
				st_ecd_cmd.meldungen.sm_reset := TRUE;
				fb_state_entry.i16_next_step := 1000;
			ELSE
				fb_soe_reset.Execute := FALSE;
				fb_state_entry.i16_next_step := 23;
			END_IF
		END_IF
	23:
		IF NOT st_masterachse.Status.DriveDeviceError THEN
			fb_ton_cmd_timeout.IN := FALSE;
			fb_state_entry.i16_next_step := 24;
		END_IF
	24:	(* Reset NC-Achsfehler *)
		CASE i16_achstyp OF
			LINEAR, RUND, LINEAR_VIRTUELL, RUND_VIRTUELL:
				IF NOT st_masterachse.Status.Error THEN
					fb_state_entry.i16_next_step := 26;
				ELSE
					fb_ton_cmd_timeout.IN := TRUE;
					mc_reset_axis.Execute := TRUE;
					IF mc_reset_axis.Busy THEN
						fb_state_entry.i16_next_step := 25;
					END_IF
				END_IF
			SERVOKLEMME7201:
				IF NOT st_masterachse.Status.Error AND NOT st_masterachse.Status.DriveDeviceError THEN
					fb_state_entry.i16_next_step := 26;
				ELSE
					fb_ton_cmd_timeout.IN := TRUE;
					mc_reset_axis.Execute := TRUE;
					IF mc_reset_axis.Busy THEN
						fb_state_entry.i16_next_step := 25;
					END_IF
				END_IF
		END_CASE
	25:
		IF NOT st_masterachse.Status.Error THEN
			mc_reset_axis.Execute := FALSE;
			fb_ton_cmd_timeout.IN := FALSE;
			fb_state_entry.i16_next_step := 26;
		END_IF
	26:
		IF st_ecd_cmd.enu_cmd = RESET THEN
			fb_state_entry.i16_next_step := 999;
		ELSE
			fb_state_entry.i16_next_step := 30;
		END_IF

(*=======================================================*)
	30:	(* Power ON NC-Achse *)
		CASE i16_achstyp OF
			LINEAR, RUND:
				fb_ton_cmd_timeout.IN := TRUE;
				IF	(st_ecd_cmd.enu_cmd > POWER_DISABLE AND st_ecd_cmd.enu_cmd < HALT_AXIS)  AND
					(NOT st_masterachse.Status.Operational OR
					(st_ecd_cmd.enu_cmd = POWER_ENABLE AND NOT st_masterachse.Status.Operational))
					THEN
						fb_state_entry.i16_next_step := 31;
				ELSE
					fb_ton_cmd_timeout.IN := FALSE;
					fb_state_entry.i16_next_step := 40;
				END_IF
			LINEAR_VIRTUELL, RUND_VIRTUELL, SERVOKLEMME7201:
				IF	st_ecd_cmd.enu_cmd > POWER_DISABLE AND st_ecd_cmd.enu_cmd < HALT_AXIS AND
					NOT mc_power_axis.Status
					THEN
						fb_state_entry.i16_next_step := 31;
				ELSE
					fb_ton_cmd_timeout.IN := FALSE;
					fb_state_entry.i16_next_step := 40;
				END_IF
		END_CASE
	31:
		mc_power_axis.Enable_Positive := TRUE;
		mc_power_axis.Enable_Negative := TRUE;
		mc_power_axis.Enable := TRUE;
		IF mc_power_axis.Busy THEN
			fb_ton_vz.PT := t#1s;
			fb_ton_vz.IN := TRUE;
			fb_state_entry.i16_next_step := 32;
		END_IF
	32:
		IF mc_power_axis.Status AND st_masterachse.Status.Operational  THEN
			IF st_ecd_cmd.enu_cmd = POWER_ENABLE THEN
				fb_state_entry.i16_next_step := 999;
			ELSE
				fb_ton_cmd_timeout.IN := FALSE;
				fb_state_entry.i16_next_step := 40;
			END_IF
		ELSIF mc_power_axis.Error AND fb_ton_vz.Q THEN
			st_ecd_cmd.meldungen.sm_power_enable := TRUE;
			err_id := mc_power_axis.ErrorID;
			fb_state_entry.i16_next_step := 1000;
		END_IF
		IF st_ecd_cmd.enu_cmd = HALT_AXIS THEN
			fb_ton_cmd_timeout.IN := FALSE;
			fb_ton_vz.IN := FALSE;
			fb_state_entry.i16_next_step := 121;
		END_IF
		IF st_ecd_cmd.enu_cmd = STOP_AXIS THEN
			fb_ton_cmd_timeout.IN := FALSE;
			fb_ton_vz.IN := FALSE;
			fb_state_entry.i16_next_step := 131;
		END_IF

(*=======================================================*)
	40:	(* Abfrage Referenzieren und Ref-Art *)
		IF st_ecd_cmd.enu_cmd = HOME THEN
			IF b_refsensor_vorhanden THEN
				mc_referenzmodus := MC_DefaultHoming;
			ELSE
				mc_referenzmodus := MC_Direct;
			END_IF
			st_position.r_referenz := 0.0;
			fb_state_entry.i16_next_step := 41;
		ELSE
			fb_ton_cmd_timeout.IN := FALSE;
			fb_state_entry.i16_next_step := 50;
		END_IF
	41:	(* Start Homing *)
		mc_home_axis.Execute := TRUE;
		mc_home_axis.Options.ClearPositionLag := TRUE;
		IF mc_home_axis.Busy THEN
			fb_state_entry.i16_next_step := 42;
		END_IF
	42:
		IF mc_home_axis.Done THEN
			mc_home_axis.Execute := FALSE;
			fb_state_entry.i16_next_step := 999;
		END_IF
		IF NOT mc_home_axis.Busy AND mc_home_axis.Error THEN
			st_ecd_cmd.meldungen.sm_home := TRUE;
			err_id := mc_home_axis.ErrorID;
			fb_state_entry.i16_next_step := 1000;
		END_IF
		IF st_ecd_cmd.enu_cmd = HALT_AXIS THEN
			mc_home_axis.Execute := FALSE;
			fb_ton_cmd_timeout.IN := FALSE;
			fb_state_entry.i16_next_step := 121;
		END_IF
		IF st_ecd_cmd.enu_cmd = STOP_AXIS THEN
			mc_home_axis.Execute := FALSE;
			fb_ton_cmd_timeout.IN := FALSE;
			fb_state_entry.i16_next_step := 131;
		END_IF

(*=======================================================*)
	50:	(* Jog vorwärts *)
		IF st_ecd_cmd.enu_cmd = JOG_VORWAERTS THEN
			fb_state_entry.i16_next_step := 51;
		ELSE
			fb_state_entry.i16_next_step := 55;
		END_IF
	51:
		b_jog_vorwaerts_execute := TRUE;
		IF mc_jog_axis.Active THEN
			fb_state_entry.i16_next_step := 52;
		ELSIF mc_jog_axis.Error THEN
			st_ecd_cmd.meldungen.sm_jog_vorwaerts := TRUE;
			fb_state_entry.i16_next_step := FEHLER;
		END_IF
	52:
		IF st_ecd_cmd.enu_cmd = JOG_STOP OR st_ecd_cmd.enu_cmd = JOG_RUECKWAERTS THEN
			fb_state_entry.i16_next_step := 61;
		END_IF

		IF st_ecd_cmd.enu_cmd = HALT_AXIS THEN
			mc_movemodulo_axis.Execute := FALSE;
			fb_ton_cmd_timeout.IN := FALSE;
			fb_state_entry.i16_next_step := 121;
		END_IF
		IF st_ecd_cmd.enu_cmd = STOP_AXIS THEN
			mc_movemodulo_axis.Execute := FALSE;
			fb_ton_cmd_timeout.IN := FALSE;
			fb_state_entry.i16_next_step := 131;
		END_IF

(*=======================================================*)
	55:	(* Jog rückwärts *)
		IF st_ecd_cmd.enu_cmd = JOG_RUECKWAERTS THEN
			fb_state_entry.i16_next_step := 56;
		ELSE
			fb_state_entry.i16_next_step := 60;
		END_IF

	56:
		b_jog_rueckwaerts_execute := TRUE;
		IF mc_jog_axis.Active THEN
			fb_state_entry.i16_next_step := 57;
		ELSIF mc_jog_axis.Error THEN
			st_ecd_cmd.meldungen.sm_jog_rueckwaerts := TRUE;
			fb_state_entry.i16_next_step := FEHLER;
		END_IF
	57:
		IF st_ecd_cmd.enu_cmd = JOG_STOP OR st_ecd_cmd.enu_cmd = JOG_VORWAERTS THEN
			fb_state_entry.i16_next_step := 61;
		END_IF

		IF st_ecd_cmd.enu_cmd = HALT_AXIS THEN
			mc_movemodulo_axis.Execute := FALSE;
			fb_ton_cmd_timeout.IN := FALSE;
			fb_state_entry.i16_next_step := 121;
		END_IF
		IF st_ecd_cmd.enu_cmd = STOP_AXIS THEN
			mc_movemodulo_axis.Execute := FALSE;
			fb_ton_cmd_timeout.IN := FALSE;
			fb_state_entry.i16_next_step := 131;
		END_IF

(*=======================================================*)
	60:	(* Jog Stop *)
		IF st_ecd_cmd.enu_cmd = JOG_STOP THEN
			fb_state_entry.i16_next_step := 61;
		ELSE
			fb_state_entry.i16_next_step := 70;
		END_IF
	61:
		b_jog_vorwaerts_execute := FALSE;
		b_jog_rueckwaerts_execute := FALSE;
		fb_state_entry.i16_next_step := 999;

(*=======================================================*)
	70:	(* Move absolute *)
		IF st_ecd_cmd.enu_cmd = MOVE_ABSOLUTE THEN
			fb_state_entry.i16_next_step := 71;
		ELSE
			fb_state_entry.i16_next_step := 80;
		END_IF
	71:
		IF ABS(st_masterachse.NcToPlc.ActPos -  st_position.r_soll ) < 0.05 THEN
			fb_state_entry.i16_next_step := 999;
		ELSE
			mc_moveabsolute_axis.Execute := TRUE;
		END_IF
		IF mc_moveabsolute_axis.Busy THEN
			fb_state_entry.i16_next_step := 72;
		END_IF
	72:
		IF mc_moveabsolute_axis.Done THEN
			mc_moveabsolute_axis.Execute := FALSE;
			fb_state_entry.i16_next_step := 999;
		END_IF
		IF NOT mc_moveabsolute_axis.Busy AND mc_moveabsolute_axis.Error THEN
			st_ecd_cmd.meldungen.sm_move_absolute := TRUE;
			err_id := mc_moveabsolute_axis.ErrorID;
			fb_state_entry.i16_next_step := 1000;
		END_IF
		IF st_ecd_cmd.enu_cmd = HALT_AXIS THEN
			mc_moveabsolute_axis.Execute := FALSE;
			fb_ton_cmd_timeout.IN := FALSE;
			fb_state_entry.i16_next_step := 121;
		END_IF
		IF st_ecd_cmd.enu_cmd = STOP_AXIS THEN
			mc_moveabsolute_axis.Execute := FALSE;
			fb_ton_cmd_timeout.IN := FALSE;
			fb_state_entry.i16_next_step := 131;
		END_IF

		(* Move-Kommando für folgende Bewegung *)
		IF st_ecd_cmd.enu_cmd = MOVE_ABSOLUTE_NEXT THEN
			fb_state_entry.i16_next_step := 74;
		END_IF
	74:
		IF ABS(st_masterachse.NcToPlc.ActPos -  st_position.r_soll ) < 0.05 THEN
			fb_state_entry.i16_next_step := 999;
		ELSE
			mc_moveabsolutenext_axis.Execute := TRUE;
		END_IF
		IF mc_moveabsolutenext_axis.Busy THEN
			fb_state_entry.i16_next_step := 75;
		END_IF
	75:
		IF mc_moveabsolutenext_axis.Done THEN
			mc_moveabsolute_axis.Execute := FALSE;
			mc_moveabsolutenext_axis.Execute := FALSE;
			fb_state_entry.i16_next_step := 999;
		END_IF
		IF NOT mc_moveabsolutenext_axis.Busy AND mc_moveabsolutenext_axis.Error THEN
			st_ecd_cmd.meldungen.sm_move_absolute := TRUE;
			err_id := mc_moveabsolutenext_axis.ErrorID;
			fb_state_entry.i16_next_step := 1000;
		END_IF
		IF st_ecd_cmd.enu_cmd = HALT_AXIS THEN
			mc_moveabsolute_axis.Execute := FALSE;
			mc_moveabsolutenext_axis.Execute := FALSE;
			fb_ton_cmd_timeout.IN := FALSE;
			fb_state_entry.i16_next_step := 121;
		END_IF
		IF st_ecd_cmd.enu_cmd = STOP_AXIS THEN
			mc_moveabsolute_axis.Execute := FALSE;
			mc_moveabsolutenext_axis.Execute := FALSE;
			fb_ton_cmd_timeout.IN := FALSE;
			fb_state_entry.i16_next_step := 131;
		END_IF

(*=======================================================*)
	80:	(* Move relative *)
		IF st_ecd_cmd.enu_cmd = MOVE_RELATIVE THEN
			fb_state_entry.i16_next_step := 81;
		ELSE
			fb_state_entry.i16_next_step := 90;
		END_IF
	81:
		mc_moverelative_axis.Execute := TRUE;
		IF mc_moverelative_axis.Busy THEN
			fb_state_entry.i16_next_step := 82;
		END_IF
	82:
		IF mc_moverelative_axis.Done THEN
			mc_moverelative_axis.Execute := FALSE;
			fb_state_entry.i16_next_step := 999;
		END_IF
		IF NOT mc_moverelative_axis.Busy AND mc_moverelative_axis.Error THEN
			st_ecd_cmd.meldungen.sm_move_relative := TRUE;
			err_id := mc_moverelative_axis.ErrorID;
			fb_state_entry.i16_next_step := 1000;
		END_IF
		IF st_ecd_cmd.enu_cmd = HALT_AXIS THEN
			mc_moverelative_axis.Execute := FALSE;
			fb_ton_cmd_timeout.IN := FALSE;
			fb_state_entry.i16_next_step := 121;
		END_IF
		IF st_ecd_cmd.enu_cmd = STOP_AXIS THEN
			mc_moverelative_axis.Execute := FALSE;
			fb_ton_cmd_timeout.IN := FALSE;
			fb_state_entry.i16_next_step := 131;
		END_IF

(*=======================================================*)
	90:	(* Move velocity *)
		IF st_ecd_cmd.enu_cmd = MOVE_VELOCITY THEN
			fb_state_entry.i16_next_step := 91;
		ELSE
			fb_state_entry.i16_next_step := 100;
		END_IF
	91:
		mc_movevelocity_axis.Execute := TRUE;
		IF mc_movevelocity_axis.Busy THEN
			fb_state_entry.i16_next_step := 92;
		END_IF
	92:
		IF mc_movevelocity_axis.InVelocity THEN
			mc_movevelocity_axis.Execute := FALSE;
			fb_state_entry.i16_next_step := 999;
		END_IF
		IF NOT mc_movevelocity_axis.Busy AND mc_movevelocity_axis.Error THEN
			st_ecd_cmd.meldungen.sm_move_velocity := TRUE;
			err_id := mc_movevelocity_axis.ErrorID;
			fb_state_entry.i16_next_step := 1000;
		END_IF
		IF st_ecd_cmd.enu_cmd = HALT_AXIS THEN
			mc_movevelocity_axis.Execute := FALSE;
			fb_ton_cmd_timeout.IN := FALSE;
			fb_state_entry.i16_next_step := 121;
		END_IF
		IF st_ecd_cmd.enu_cmd = STOP_AXIS THEN
			mc_movevelocity_axis.Execute := FALSE;
			fb_ton_cmd_timeout.IN := FALSE;
			fb_state_entry.i16_next_step := 131;
		END_IF

(*=======================================================*)
	100:	(* Move modulo *)
		IF st_ecd_cmd.enu_cmd = MOVE_MODULO THEN
			fb_state_entry.i16_next_step := 101;
		ELSE
			fb_state_entry.i16_next_step := 103;
		END_IF
	101:
		IF ABS(st_masterachse.NcToPlc.ModuloActPos -  st_position.r_soll ) < 0.3 THEN
			fb_state_entry.i16_next_step := 999;
		ELSE
			mc_movemodulo_axis.Execute := TRUE;
		END_IF
		IF mc_movemodulo_axis.Busy THEN
			fb_state_entry.i16_next_step := 102;
		END_IF
	102:
		IF mc_movemodulo_axis.Done THEN
			mc_movemodulo_axis.Execute := FALSE;
			fb_state_entry.i16_next_step := 999;
		END_IF

		IF NOT mc_movemodulo_axis.Busy AND mc_movemodulo_axis.Error THEN
			st_ecd_cmd.meldungen.sm_move_modulo := TRUE;
			err_id := mc_movemodulo_axis.ErrorID;
			fb_state_entry.i16_next_step := 1000;
		END_IF
		IF st_ecd_cmd.enu_cmd = HALT_AXIS THEN
			mc_movemodulo_axis.Execute := FALSE;
			fb_ton_cmd_timeout.IN := FALSE;
			fb_state_entry.i16_next_step := 121;
		END_IF
		IF st_ecd_cmd.enu_cmd = STOP_AXIS THEN
			mc_movemodulo_axis.Execute := FALSE;
			fb_ton_cmd_timeout.IN := FALSE;
			fb_state_entry.i16_next_step := 131;
		END_IF

(*=======================================================*)
	103:
		(*Touch Probe checken*)
		IF	fb_state_entry.E THEN
			mc_abort_trigger.Execute:=TRUE;
		END_IF

		IF st_ecd_cmd.enu_cmd = MOVE_TOUCH_PROBE THEN

			(*Touch Probe darf nicht betätigt sein*)
			IF	(b_FallingEdge AND NOT b_TriggerInput) OR
				(NOT b_FallingEdge AND b_TriggerInput)  THEN
				st_ecd_cmd.meldungen.sm_touch_probe_defect := TRUE;		(*Messtaster defekt*)
				fb_state_entry.i16_next_step := FEHLER;

			ELSIF mc_abort_trigger.Done THEN
				lr_RecPos:=0;
				fb_state_entry.i16_next_step := 104;
			END_IF

		ELSE
			fb_state_entry.i16_next_step := 110;
		END_IF

		IF	fb_state_entry.X THEN
			mc_abort_trigger.Execute:=FALSE;
		END_IF

	104:
		(* Move absolute (Position muss hinter dem Touch Probe liegen => der Restweg wird gelöscht)*)
		IF 	ABS(st_masterachse.NcToPlc.ActPos -  st_position.r_soll ) < 0.05 THEN
			fb_state_entry.i16_next_step := 999;
		ELSE
			mc_moveabsolute_axis.Execute := TRUE;
			mc_touch_probe.Execute:=TRUE;
		END_IF
		IF 	mc_moveabsolute_axis.Busy THEN
			fb_state_entry.i16_next_step := 105;
		END_IF

	105:
		(*Achsposition wurde erreicht ohne Taster Event*)
		IF 	mc_moveabsolute_axis.Done THEN
			fb_state_entry.i16_next_step := 999;
		END_IF

		(*Achse anhalten wenn Touch Probe betätigt wird*)
		IF 	mc_moveabsolute_axis.Busy AND
			(b_TriggerInput = NOT b_FallingEdge OR
			mc_touch_probe.Done) THEN
			fb_state_entry.i16_next_step := 131;
		END_IF

		(*Übergabe Rec Position*)
		IF	mc_touch_probe.Done THEN
			lr_RecPos:=mc_touch_probe.RecordedPosition;
		END_IF

		(*Fehler Achse*)
		IF 	NOT mc_moveabsolute_axis.Busy AND mc_moveabsolute_axis.Error THEN
			st_ecd_cmd.meldungen.sm_move_absolute := TRUE;
			err_id := mc_moveabsolute_axis.ErrorID;
			fb_state_entry.i16_next_step := FEHLER;
		END_IF

		(*Fehler Touch Probe*)
		IF  	mc_touch_probe.Error THEN
			st_ecd_cmd.meldungen.sm_touch_probe_err := TRUE;
			err_id := mc_touch_probe.ErrorID;
			fb_state_entry.i16_next_step := FEHLER;
		END_IF

		IF	fb_state_entry.X THEN
			fb_ton_cmd_timeout.IN := FALSE;
			mc_moveabsolute_axis.Execute := FALSE;
			mc_touch_probe.Execute:=FALSE;
		END_IF

(*=======================================================*)
	110:	(* Position *)
		IF st_ecd_cmd.enu_cmd = SET_POSITION THEN
			fb_state_entry.i16_next_step := 111;
		ELSE
			fb_state_entry.i16_next_step := 121;
		END_IF
	111:
		(* Soll- und Istposition werden auf den gleichen Wert gesetzt und somit der Schleppfehler gelöscht. *)
		mc_setposition_axis.Options.ClearPositionLag := TRUE;
		mc_setposition_axis.Options.EncoderIndex := 0;
		mc_setposition_axis.Options.SelectEncoderIndex := FALSE;
		mc_setposition_axis.Execute := TRUE;
		IF mc_setposition_axis.Busy THEN
			fb_state_entry.i16_next_step := 112;
		END_IF
	112:
		IF mc_setposition_axis.Done THEN
			mc_setposition_axis.Execute := FALSE;
			fb_state_entry.i16_next_step := 999;
		END_IF
		IF NOT mc_setposition_axis.Busy AND mc_setposition_axis.Error THEN
			st_ecd_cmd.meldungen.sm_setposition := TRUE;
			err_id := mc_setposition_axis.ErrorID;
			fb_state_entry.i16_next_step := 1000;
		END_IF
		IF st_ecd_cmd.enu_cmd = HALT_AXIS THEN
			mc_setposition_axis.Execute := FALSE;
			fb_ton_cmd_timeout.IN := FALSE;
			fb_state_entry.i16_next_step := 121;
		END_IF
		IF st_ecd_cmd.enu_cmd = STOP_AXIS THEN
			mc_setposition_axis.Execute := FALSE;
			fb_ton_cmd_timeout.IN := FALSE;
			fb_state_entry.i16_next_step := 131;
		END_IF

(*=======================================================*)
	120:	(* Halt *)
		fb_ton_cmd_timeout.IN := TRUE;
		IF st_ecd_cmd.enu_cmd = HALT_AXIS THEN
			fb_state_entry.i16_next_step := 121;
		ELSE
			fb_ton_cmd_timeout.IN := FALSE;
			fb_state_entry.i16_next_step := 131;
		END_IF
	121:
		mc_halt_axis.Execute := TRUE;
		IF mc_halt_axis.Busy THEN
			fb_state_entry.i16_next_step := 122;
		END_IF
	122:
		IF mc_halt_axis.Done THEN
			mc_halt_axis.Execute := FALSE;
			fb_state_entry.i16_next_step := 123;
		END_IF
		IF NOT mc_halt_axis.Busy AND mc_halt_axis.Error THEN
			st_ecd_cmd.meldungen.sm_halt_axis := TRUE;
			err_id := mc_halt_axis.ErrorID;
			fb_state_entry.i16_next_step := 1000;
		END_IF
	123:
		IF	NOT st_masterachse.Status.ConstantVelocity AND
			NOT st_masterachse.Status.Accelerating AND
			NOT st_masterachse.Status.Decelerating
			THEN
				fb_state_entry.i16_next_step := 999;
		END_IF

(*=======================================================*)
	130: (* Stop *)
		fb_ton_cmd_timeout.IN := TRUE;
		IF st_ecd_cmd.enu_cmd = STOP_AXIS THEN
			fb_state_entry.i16_next_step := 131;
		ELSE
			fb_ton_cmd_timeout.IN := FALSE;
			fb_state_entry.i16_next_step := 140;
		END_IF
	131:
		mc_stop_axis.Execute := TRUE;
		IF mc_stop_axis.Busy THEN
			fb_state_entry.i16_next_step := 132;
		END_IF
	132:
		IF mc_stop_axis.Done THEN
			mc_stop_axis.Execute := FALSE;
			fb_state_entry.i16_next_step := 133;
		END_IF
		IF mc_stop_axis.Error THEN
			st_ecd_cmd.meldungen.sm_stop_axis := TRUE;
			err_id := mc_stop_axis.ErrorID;
			fb_state_entry.i16_next_step := 1000;
		END_IF
	133:
		IF 	NOT st_masterachse.Status.ConstantVelocity AND
			NOT st_masterachse.Status.Accelerating AND
			NOT st_masterachse.Status.Decelerating
			THEN
				fb_state_entry.i16_next_step := 999;
		END_IF

(*=======================================================*)
	140:	(* Frei *)
		fb_state_entry.i16_next_step := 500;

(*======================Parameterbefehle=================================*)
	500:	(* Schreibe einen Parameter an den Antrieb *)
		fb_ton_cmd_timeout.IN := TRUE;
		IF st_ecd_cmd.enu_cmd = SOE_WRITE_PARAM THEN
			fb_state_entry.i16_next_step := 501;
		ELSE
			fb_ton_cmd_timeout.IN := FALSE;
			fb_state_entry.i16_next_step := 510;
		END_IF
	501:
		fb_soe_write.Execute := TRUE;
		IF fb_soe_write.Busy THEN
			fb_state_entry.i16_next_step := 502;
		END_IF
	502:
		IF NOT fb_soe_write.Busy THEN
			fb_soe_write.Execute := FALSE;
			IF fb_soe_write.Error THEN
				st_ecd_cmd.meldungen.sm_write_soe_parameter := TRUE;
				fb_state_entry.i16_next_step := 1000;
			ELSE
				fb_state_entry.i16_next_step := 999;
			END_IF
		END_IF

(*=======================================================*)
	510:	(* Lesen eines Parameter vom Antrieb *)
		fb_ton_cmd_timeout.IN := TRUE;
		IF st_ecd_cmd.enu_cmd = SOE_READ_PARAM THEN
			fb_state_entry.i16_next_step := 511;
		ELSE
			fb_ton_cmd_timeout.IN := FALSE;
			fb_state_entry.i16_next_step := 520;
		END_IF
	511:
		fb_soe_read.Execute := TRUE;
		IF fb_soe_read.Busy THEN
			fb_state_entry.i16_next_step := 512;
		END_IF
	512:
		IF NOT fb_soe_read.Busy THEN
			fb_soe_write.Execute := FALSE;
			IF fb_soe_read.Error THEN
				st_ecd_cmd.meldungen.sm_read_soe_parameter := TRUE;
				fb_state_entry.i16_next_step := 1000;
			ELSE
				fb_state_entry.i16_next_step := 999;
			END_IF
		END_IF

(*=======================================================*)
	520:	(* Schreibe einen Parameter an die NC-Achse *)
		fb_ton_cmd_timeout.IN := TRUE;
		IF st_ecd_cmd.enu_cmd = WRITE_NC_PARAMETER THEN
			fb_state_entry.i16_next_step := 521;
		ELSE
			fb_ton_cmd_timeout.IN := FALSE;
			fb_state_entry.i16_next_step := 530;
		END_IF
	521:
		mc_write_nc_parameter.Execute := TRUE;
		IF mc_write_nc_parameter.Busy THEN
			fb_state_entry.i16_next_step := 522;
		END_IF
	522:
		IF NOT mc_write_nc_parameter.Busy THEN
			mc_write_nc_parameter.Execute := FALSE;
			IF mc_write_nc_parameter.Error THEN
				st_ecd_cmd.meldungen.sm_write_nc_parameter := TRUE;
				fb_state_entry.i16_next_step := 1000;
			ELSE
				fb_state_entry.i16_next_step := 999;
			END_IF
		END_IF

(*=======================================================*)
	530:	(* Lesen eines Parameter vom der NC-Achse *)
		fb_ton_cmd_timeout.IN := TRUE;
		IF st_ecd_cmd.enu_cmd = READ_NC_PARAMETER THEN
			fb_state_entry.i16_next_step := 531;
		ELSE
			fb_ton_cmd_timeout.IN := FALSE;
			fb_state_entry.i16_next_step := 540;
		END_IF
	531:
		mc_read_nc_parameter.Enable := TRUE;
		IF mc_read_nc_parameter.Busy THEN
			fb_state_entry.i16_next_step := 532;
		END_IF
	532:
		IF NOT mc_read_nc_parameter.Busy THEN
			mc_read_nc_parameter.Enable := FALSE;
			IF mc_read_nc_parameter.Error THEN
				st_ecd_cmd.meldungen.sm_read_nc_parameter := TRUE;
				fb_state_entry.i16_next_step := 1000;
			ELSE
				fb_state_entry.i16_next_step := 999;
			END_IF
		END_IF

(*=======================================================*)
	540:	(* Schreibe einen beliebigen ADS-Parameter an die NC-Achse *)
		fb_ton_cmd_timeout.IN := TRUE;
		IF st_ecd_cmd.enu_cmd = WRITE_ADS_PARAMETER THEN
			fb_state_entry.i16_next_step := 541;
		ELSE
			fb_ton_cmd_timeout.IN := FALSE;
			fb_state_entry.i16_next_step := 550;
		END_IF
	541:
		fb_ads_write.WRITE := TRUE;
		IF fb_ads_write.BUSY THEN
			fb_state_entry.i16_next_step := 542;
		END_IF
	542:
		IF NOT fb_ads_write.BUSY THEN
			fb_ads_write.WRITE := FALSE;
			IF fb_ads_write.ERR THEN
				st_ecd_cmd.meldungen.sm_write_ads_parameter := TRUE;
				fb_state_entry.i16_next_step := 1000;
			ELSE
				fb_state_entry.i16_next_step := 999;
			END_IF
		END_IF

(*=======================================================*)
	550:	(* Lesen einen beliebigenADS-Parameter vom der NC-Achse *)
		fb_ton_cmd_timeout.IN := TRUE;
		IF st_ecd_cmd.enu_cmd = READ_ADS_PARAMETER THEN
			fb_state_entry.i16_next_step := 551;
		ELSE
			fb_ton_cmd_timeout.IN := FALSE;
			fb_state_entry.i16_next_step := 560;
		END_IF
	551:
		fb_ads_read.READ := TRUE;
		IF fb_ads_read.BUSY THEN
			fb_state_entry.i16_next_step := 552;
		END_IF
	552:
		IF NOT fb_ads_read.BUSY THEN
			fb_ads_read.READ := FALSE;
			IF fb_ads_read.ERR THEN
				st_ecd_cmd.meldungen.sm_read_ads_parameter := TRUE;
				fb_state_entry.i16_next_step := 1000;
			ELSE
				fb_state_entry.i16_next_step := 999;
			END_IF
		END_IF

(*=======================================================*)
	560:	(* Schreibe die neuen EcSoe Parameter an den Antrieb *)
		fb_ton_cmd_timeout.IN := TRUE;
		IF st_ecd_cmd.enu_cmd = ECCOESDO_WRITE_PARAM THEN
			fb_state_entry.i16_next_step := 561;
		ELSE
			fb_ton_cmd_timeout.IN := FALSE;
			fb_state_entry.i16_next_step := 570;
		END_IF
	561:
		fb_ec_coe_sdo_write_ex.bExecute := TRUE;
		IF fb_ec_coe_sdo_write_ex.bBusy THEN
			fb_state_entry.i16_next_step := 562;
		END_IF
	562:
		IF NOT fb_ec_coe_sdo_write_ex.bBusy THEN
			fb_ec_coe_sdo_write_ex.bExecute := FALSE;
			IF fb_ec_coe_sdo_write_ex.bError THEN
				st_ecd_cmd.meldungen.sm_ec_coe_sdo_write_ex := TRUE;
				fb_state_entry.i16_next_step := 1000;
			ELSE
				fb_state_entry.i16_next_step := 999;
			END_IF
		END_IF

(*=======================================================*)
	570:	(* Lese die neuen EcSoe Parameter an den Antrieb *)
		fb_ton_cmd_timeout.IN := TRUE;
		IF st_ecd_cmd.enu_cmd = ECCOESDO_READ_PARAM THEN
			fb_state_entry.i16_next_step := 571;
		ELSE
			fb_ton_cmd_timeout.IN := FALSE;
			fb_state_entry.i16_next_step := 580;
		END_IF
	571:
		fb_ec_coe_sdo_read_ex.bExecute := TRUE;
		IF fb_ec_coe_sdo_read_ex.bBusy THEN
			fb_state_entry.i16_next_step := 572;
		END_IF
	572:
		IF NOT fb_ec_coe_sdo_read_ex.bBusy THEN
			fb_ec_coe_sdo_read_ex.bExecute := FALSE;
			IF fb_ec_coe_sdo_read_ex.bError THEN
				st_ecd_cmd.meldungen.sm_ec_coe_sdo_read_ex := TRUE;
				fb_state_entry.i16_next_step := 1000;
			ELSE
				fb_state_entry.i16_next_step := 999;
			END_IF
		END_IF

(*=======================================================*)
	580:	(* Frei *)
		fb_state_entry.i16_next_step := 999;

(*=======================================================*)
	999:	(* Ende - Befehl wurde korrekt abgearbeitet *)
		st_ecd_cmd.enu_cmd := NO_COMMAND;
		fb_ton_cmd_timeout.IN := FALSE;
		fb_ton_vz.IN := FALSE;

		b_jog_vorwaerts_execute := FALSE;
		b_jog_rueckwaerts_execute := FALSE;

		mc_reset_axis.Execute := FALSE;
		mc_home_axis.Execute := FALSE;
		mc_moveabsolute_axis.Execute := FALSE;
		mc_moverelative_axis.Execute := FALSE;
		mc_movevelocity_axis.Execute := FALSE;
		mc_movemodulo_axis.Execute := FALSE;
		mc_setposition_axis.Execute := FALSE;
		mc_halt_axis.Execute := FALSE;
		mc_stop_axis.Execute := FALSE;
		fb_soe_reset.Execute := FALSE;
		fb_soe_write.Execute := FALSE;
		fb_soe_read.Execute := FALSE;
		mc_write_nc_parameter.Execute := FALSE;
		mc_read_nc_parameter.Enable := FALSE;
		fb_ads_write.WRITE := FALSE;
		fb_ads_read.READ := FALSE;
		fb_ec_coe_sdo_write_ex.bExecute := FALSE;
		fb_ec_coe_sdo_read_ex.bExecute := FALSE;

		st_ecd_cmd.meldungen.sm_power_enable := FALSE;
		st_ecd_cmd.meldungen.sm_power_disable := FALSE;
		st_ecd_cmd.meldungen.sm_reset := FALSE;
		st_ecd_cmd.meldungen.sm_home := FALSE;
		st_ecd_cmd.meldungen.sm_setposition := FALSE;
		st_ecd_cmd.meldungen.sm_jog_vorwaerts := FALSE;
		st_ecd_cmd.meldungen.sm_jog_rueckwaerts := FALSE;
		st_ecd_cmd.meldungen.sm_move_absolute := FALSE;
		st_ecd_cmd.meldungen.sm_move_relative := FALSE;
		st_ecd_cmd.meldungen.sm_move_velocity := FALSE;
		st_ecd_cmd.meldungen.sm_move_modulo := FALSE;
		st_ecd_cmd.meldungen.sm_stop_axis := FALSE;
		st_ecd_cmd.meldungen.sm_halt_axis := FALSE;
		st_ecd_cmd.meldungen.sm_motion_command_timeout := FALSE;
		st_ecd_cmd.meldungen.sm_limit_positiv_erreicht := FALSE;
		st_ecd_cmd.meldungen.sm_limit_negativ_erreicht := FALSE;
		st_ecd_cmd.meldungen.sm_write_soe_parameter := FALSE;
		st_ecd_cmd.meldungen.sm_read_soe_parameter := FALSE;
		st_ecd_cmd.meldungen.sm_write_nc_parameter := FALSE;
		st_ecd_cmd.meldungen.sm_read_nc_parameter := FALSE;
		st_ecd_cmd.meldungen.sm_write_ads_parameter := FALSE;
		st_ecd_cmd.meldungen.sm_read_ads_parameter := FALSE;
		st_ecd_cmd.meldungen.sm_ec_coe_sdo_write_ex := FALSE;
		st_ecd_cmd.meldungen.sm_ec_coe_sdo_read_ex := FALSE;

		fb_state_entry.i16_next_step := 1;

(*=======================================================*)
	1000: (* Fehler *)
		IF fb_state_entry.E THEN
			st_ecd_cmd.b_job_fehler := TRUE;
			fb_ton_cmd_timeout.IN := FALSE;
			fb_ton_vz.IN := FALSE;
			st_ecd_cmd.enu_cmd := NO_COMMAND;
		END_IF

		(* Fehler reseten *)
		IF st_ecd_cmd.enu_cmd >= ABORT THEN
			st_ecd_cmd.b_job_fehler := FALSE;
			b_jog_vorwaerts_execute := FALSE;
			b_jog_rueckwaerts_execute := FALSE;
			mc_reset_axis.Execute := FALSE;
			mc_home_axis.Execute := FALSE;
			mc_moveabsolute_axis.Execute := FALSE;
			mc_moverelative_axis.Execute := FALSE;
			mc_movevelocity_axis.Execute := FALSE;
			mc_movemodulo_axis.Execute := FALSE;
			mc_setposition_axis.Execute := FALSE;
			mc_halt_axis.Execute := FALSE;
			mc_stop_axis.Execute := FALSE;
			fb_soe_reset.Execute := FALSE;
			fb_soe_write.Execute := FALSE;
			fb_soe_read.Execute := FALSE;
			mc_write_nc_parameter.Execute := FALSE;
			mc_read_nc_parameter.Enable := FALSE;
			fb_ads_write.WRITE := FALSE;
			fb_ads_read.READ := FALSE;
			fb_ec_coe_sdo_write_ex.bExecute := FALSE;
			fb_ec_coe_sdo_read_ex.bExecute := FALSE;
			fb_state_entry.i16_next_step := 0;
		END_IF
END_CASE

(* Endlagenüberwachung der maximalen Verfahrwege der Achse *)
IF b_limitsensor_positiv_vorhanden AND fb_f_trig_limit_sensor_positiv.Q THEN
	mc_stop_axis.Execute := TRUE;
	st_ecd_cmd.meldungen.sm_limit_positiv_erreicht := TRUE;
	fb_state_entry.i16_next_step := 1000;
END_IF
IF b_limitsensor_negativ_vorhanden AND fb_f_trig_limit_sensor_negativ.Q THEN
	mc_stop_axis.Execute := TRUE;
	st_ecd_cmd.meldungen.sm_limit_negativ_erreicht := TRUE;
	fb_state_entry.i16_next_step := 1000;
END_IF

(* Timeout-Fehler aller Drivekommandos *)
IF fb_ton_cmd_timeout.Q THEN
	fb_ton_cmd_timeout.IN := FALSE;
	st_ecd_cmd.meldungen.sm_motion_command_timeout := TRUE;
	fb_state_entry.i16_next_step := 1000;
END_IF

(*Abbruch des aktuellen Achskommandos *)
IF st_ecd_cmd.enu_cmd = ABORT AND fb_state_entry.i16_next_step <> FEHLER THEN
	fb_state_entry.i16_next_step := 999;
END_IF

(* Statehistory *)
fb_state_entry(
	i16_next_step:= ,
	i16_pos:= 2,
	s_debugtext:= ,
	E=> , 
	X=> , 
	i16_step=> ,
	i16_last_step=> );

fb_cmd_history(i16_current_cmd:= st_ecd_cmd.enu_cmd, last_cmd=> );

(*=============================================================================================*)
(* Ab hier werden alle Verfahraufträge für eine Achse abgewickelt *)

(* Lese Zustand der Achse *)
st_masterachse.ReadStatus;

(* Für Rundachsen muss die Sollgeschwindigkeit umgerechnet werden in °/s *)
IF i16_achstyp = RUND OR i16_achstyp = RUND_VIRTUELL THEN
	lr_sollgeschwindigkeit := lr_sollgeschwindigkeit * 360 / 60;
END_IF

(*=============================================================================================*)
(* Reglerfreigabe *)
mc_power_axis(
	Enable:= ,
	Enable_Positive:= ,
	Enable_Negative:= ,
	Override:= lr_override,
	BufferMode:= mc_buffermode_axis,
	Axis:= st_masterachse,
	Status=> ,
	Busy=> ,
	Active=> ,
	Error=> ,
	ErrorID=> );

(*=============================================================================================*)
(* Achse aus Fehlerzustand rücksetzen *)
(* NC-Achse *)
mc_reset_axis(
	Execute:= ,
	Axis:= st_masterachse,
	Done=> ,
	Busy=> ,
	Error=> ,
	ErrorID=> );

(* AX5000 Servokontroller *)
fb_soe_reset(
	NetId:= , 
	Execute:= , 
	Timeout:= t_ads_timeout,
	Axis:= st_masterachse,
	Busy=> ,
	Error=> , 
	AdsErrId=> , 
	SercosErrId=> );

(*=============================================================================================*)
(* Achsposition setzen *)
mc_setposition_axis(
	Execute:= ,
	Position:= st_position.r_soll,
	Mode:= FALSE, (* RELATIVE=True, ABSOLUTE=False (Default) *)
	Options:= ,
	Axis:= st_masterachse,
	Done=> ,
	Busy=> ,
	Error=> ,
	ErrorID=> );

(*=============================================================================================*)
(* Achse referenzieren *)
mc_home_axis(
	Execute:= ,
	Position:= st_position.r_referenz,
	HomingMode:= mc_referenzmodus,
	BufferMode:= mc_buffermode_axis,
	Options:= ,
	bCalibrationCam:= e_referenznocken,
	Axis:= st_masterachse,
	Done=> ,
	Busy=> ,
	Active=> ,
	CommandAborted=> ,
	Error=> ,
	ErrorId=> );

(*=============================================================================================*)
(* Achse tippen *)
mc_jog_axis(
	JogForward:= b_jog_vorwaerts_execute AND NOT b_jog_rueckwaerts_execute,
	JogBackwards:= b_jog_rueckwaerts_execute AND NOT b_jog_vorwaerts_execute,
	Mode:= MC_JOGMODE_CONTINOUS,  (* motion with standard jog parameters for slow motion *)
	Velocity:= lr_sollgeschwindigkeit,
	Acceleration:= st_vorgabe_geschwindigkeiten.lr_beschleunigung,
	Deceleration:= st_vorgabe_geschwindigkeiten.lr_verzoegerung,
	Jerk:= st_vorgabe_geschwindigkeiten.lr_ruck,
	Axis:= st_masterachse,
	Done=> ,
	Busy=> ,
	Active=> ,
	CommandAborted=> ,
	Error=> ,
	ErrorId=> );

(*=============================================================================================*)
(* Fahre Achse absolut *)
mc_moveabsolute_axis(
	Execute:= ,
	Position:= st_position.r_soll,
	Velocity:= lr_sollgeschwindigkeit,
	Acceleration:= st_vorgabe_geschwindigkeiten.lr_beschleunigung,
	Deceleration:= st_vorgabe_geschwindigkeiten.lr_verzoegerung,
	Jerk:= st_vorgabe_geschwindigkeiten.lr_ruck,
	BufferMode:= mc_buffermode_axis,
	Options:= ,
	Axis:= st_masterachse,
	Done=> ,
	Busy=> ,
	Active=> ,
	CommandAborted=> ,
	Error=> ,
	ErrorID=> );
(* Fahre Achse absolut im Falle einer Folgebewegung *)
mc_moveabsolutenext_axis(
	Execute:= ,
	Position:= st_position.r_soll,
	Velocity:= lr_sollgeschwindigkeit,
	Acceleration:= st_vorgabe_geschwindigkeiten.lr_beschleunigung,
	Deceleration:= st_vorgabe_geschwindigkeiten.lr_verzoegerung,
	Jerk:= st_vorgabe_geschwindigkeiten.lr_ruck,
	BufferMode:= mc_buffermode_axis,
	Options:= ,
	Axis:= st_masterachse,
	Done=> ,
	Busy=> ,
	Active=> ,
	CommandAborted=> ,
	Error=> ,
	ErrorID=> );

(*=============================================================================================*)
(* Fahre Achse relaiv *)
mc_moverelative_axis(
	Execute:= ,
	Distance:= st_position.r_soll,
	Velocity:= lr_sollgeschwindigkeit,
	Acceleration:= st_vorgabe_geschwindigkeiten.lr_beschleunigung,
	Deceleration:= st_vorgabe_geschwindigkeiten.lr_verzoegerung,
	Jerk:= st_vorgabe_geschwindigkeiten.lr_ruck,
	BufferMode:= mc_buffermode_axis,
	Options:= ,
	Axis:= st_masterachse,
	Done=> ,
	Busy=> ,
	Active=> ,
	CommandAborted=> ,
	Error=> ,
	ErrorID=> );

(*=============================================================================================*)
(* Gleichlaufachse starten *)
mc_movevelocity_axis(
	Execute:= ,
	Velocity:= lr_sollgeschwindigkeit,
	Acceleration:= st_vorgabe_geschwindigkeiten.lr_beschleunigung,
	Deceleration:= st_vorgabe_geschwindigkeiten.lr_verzoegerung,
	Jerk:= st_vorgabe_geschwindigkeiten.lr_ruck,
	Direction:= mc_richtung_velocity,
	BufferMode:= mc_buffermode_axis,
	Options:= ,
	Axis:= st_masterachse,
	InVelocity=> ,
	Busy=> ,
	Active=> ,
	CommandAborted=> ,
	Error=> ,
	ErrorID=> );

(*=============================================================================================*)
(* Bewegen einer Rundachse *)
mc_movemodulo_axis(
	Execute:= ,
	Position:= st_position.r_soll,
	Velocity:= lr_sollgeschwindigkeit,
	Acceleration:= st_vorgabe_geschwindigkeiten.lr_beschleunigung,
	Deceleration:= st_vorgabe_geschwindigkeiten.lr_verzoegerung,
	Jerk:= st_vorgabe_geschwindigkeiten.lr_ruck,
	Direction:= mc_richtung_modulo,
	BufferMode:= mc_buffermode_axis,
	Options:= ,
	Axis:= st_masterachse,
	Done=> ,
	Busy=> ,
	Active=> ,
	CommandAborted=> ,
	Error=> ,
	ErrorID=> );

(*=============================================================================================*)
mc_stop_axis(
	Execute:= ,
	Deceleration:= st_vorgabe_geschwindigkeiten.lr_verzoegerung,
	Jerk:= st_vorgabe_geschwindigkeiten.lr_ruck,
	Options:= ,
	Axis:= st_masterachse,
	Done=> ,
	Busy=> ,
	Active=> ,
	CommandAborted=> ,
	Error=> ,
	ErrorID=> );

(*=============================================================================================*)
(* MC_Halt führt einen normalen Halt während der Bewegung aus.
Im Gegensatz dazu verriegelt MC_Stop die Achse gegen weitere Bewegungskommandos und
sollte nur in besonderen Situationen angewendet werden. *)
mc_halt_axis(
	Execute:= ,
	Deceleration:= st_vorgabe_geschwindigkeiten.lr_verzoegerung,
	Jerk:= st_vorgabe_geschwindigkeiten.lr_ruck,
	BufferMode:= mc_buffermode_axis,
	Options:= ,
	Axis:= st_masterachse,
	Done=> ,
	Busy=> ,
	Active=> ,
	CommandAborted=> ,
	Error=> ,
	ErrorID=> );

(*=============================================================================================*)
(* Einen Parameter auf den Antrieb schreiben *)
fb_soe_write(
	NetId:= , 
	Idn:= w_idn,	(* Idn := S_0_IDN + 33; *)
	Element:= EC_SOE_ELEMENT_VALUE,
	pSrcBuf:= ADR(ui16_soeparam_write_value),
	BufLen:= SIZEOF(ui16_soeparam_write_value),
	Execute:= , 
	Timeout:= t_ads_timeout,
	Password:= ,
	Axis:= st_masterachse,
	Busy=> ,
	Error=> ,
	AdsErrId=> ,
	SercosErrId=> );

(*=============================================================================================*)
(* Einen Parameter auf dem Antrieb lesen  *)
fb_soe_read(
	NetId:= , 
	Idn:= w_idn,	(* Idn := S_0_IDN + 33; *)
	Element:= EC_SOE_ELEMENT_VALUE,
	pDstBuf:= ADR(ui16_soeparam_read_value),
	BufLen:= SIZEOF(ui16_soeparam_read_value),
	Execute:= , 
	Timeout:= t_ads_timeout,
	Axis:= st_masterachse,
	Busy=> ,
	Error=> , 
	AdsErrId=> ,
	SercosErrId=> , 
	Attribute=> );

(*=============================================================================================*)
(* Einen Parameter auf die NC-Achse schreiben *)
mc_write_nc_parameter(
	Execute:= , 
	ParameterNumber:= i16_nc_parameter_nummer,
	Value:= r_wert_nc_write_parameter,
	Axis:= st_masterachse,
	Done=> ,
	Busy=> ,
	Error=> , 
	ErrorID=> );

(*=============================================================================================*)
(* Einen Parameter von der NC-Achse lesen *)
mc_read_nc_parameter(
	Enable:= , 
	ParameterNumber:= i16_nc_parameter_nummer,
	ReadMode:= READMODE_ONCE,
	Axis:= st_masterachse,
	Valid=> ,
	Busy=> ,
	Error=> , 
	ErrorID=> , 
	Value=> r_wert_nc_read_parameter);

(*=============================================================================================*)
(* Einen beliebigen ADS-Parameter auf die NC-Achse schreiben *)
fb_ads_write(
	NETID:= ,
	PORT:= 501,
	IDXGRP:= st_ads_info.st_symbol_info.idxGroup,
	IDXOFFS:= st_ads_info.st_symbol_info.idxOffset,
	LEN:= st_ads_info.st_symbol_info.byteSize,
	SRCADDR:= st_ads_info.dw_quelladresse_ads_write,
	WRITE:= ,
	TMOUT:= t_ads_timeout,
	BUSY=> , 
	ERR=> , 
	ERRID=> );

(*=============================================================================================*)
(* Einen beliebigen ADS-Parameter von der NC-Achse lesen *)
fb_ads_read(
	NETID:= ,
	PORT:= 501,
	IDXGRP:= st_ads_info.st_symbol_info.idxGroup,
	IDXOFFS:= st_ads_info.st_symbol_info.idxOffset,
	LEN:= st_ads_info.st_symbol_info.byteSize,
	DESTADDR:= st_ads_info.dw_zieladresse_ads_read,
	READ:= , 
	TMOUT:= t_ads_timeout,
	BUSY=> , 
	ERR=> , 
	ERRID=> );

(*=============================================================================================*)
(* Einen neuen EcCoeSdo-Parameter auf den Antrieb schreiben *)
fb_ec_coe_sdo_write_ex(
	sNetId:= st_eccoe_sdo.s_ec_slave_net_id,
	nSlaveAddr:= st_eccoe_sdo.ui16_slave_addr,
	nSubIndex:= st_eccoe_sdo.i8_sub_index,
	nIndex:= st_eccoe_sdo.w_index,
	pSrcBuf:= st_eccoe_sdo.dw_p_source_buffer,
	cbBufLen:= st_eccoe_sdo.ui32_buffer_length,
	bExecute:= ,
	tTimeout:= t_ads_timeout,
	bCompleteAccess:= FALSE,
	bBusy=> , 
	bError=> ,
	nErrId=> );

(*=============================================================================================*)
(* Einen neuen EcCoeSdo-Parameter von dem Antrieb lesen *)
fb_ec_coe_sdo_read_ex(
	sNetId:= st_eccoe_sdo.s_ec_slave_net_id,
	nSlaveAddr:= st_eccoe_sdo.ui16_slave_addr,
	nSubIndex:= st_eccoe_sdo.i8_sub_index,
	nIndex:= st_eccoe_sdo.w_index,
	pDstBuf:= st_eccoe_sdo.dw_p_destination_buffer,
	cbBufLen:= st_eccoe_sdo.ui32_buffer_length,
	bExecute:= ,
	tTimeout:= t_ads_timeout,
	bCompleteAccess:= FALSE,
	bBusy=> ,
	bError=> ,
	nErrId=> );
END_FUNCTION_BLOCK
ACTION sub_TouchProbe:
(*======================================================
   Command: MOVE_TOUCH_PROBE
 ------------------------------------------------------
   Auth: 		Werner Friedl    						 
   Date: 		10.09.2019    						     
   Rev.: 		1.0	
   Desc:		Mit diesem Command kann die Achsposition zu eimem Tastzeitpunkt aufgezeichnet werden.

			- im Achsaufruf müssen diese Einstellungen gemacht werden
		z.B.		b_TriggerInput:=i16_DigitalInput.0		=> Verknüpfung mit den Prozessdaten der Achse an dem der Taster angeklemmt wurde				
				i16_TouchProbeInNo:=1					=> 1 wenn der Taster am Input 1 angeklemmt wurde
				b_SignalEdge:=FallingEdge				=> FallingEdge ODER RisingEdge

		- das Kommando MOVE_TOUCH_PROBE fährt die Achse auf den Taster. Wird der Taster 
			während der Fahrt betätigt , dann stoppt die Achse automatisch und 
			das Messergebniss landet in der VAR lr_RecPos
		
		- Schritt103 => Taster prüfen
		- Schritt104 => Move Absolut und start Touch Probe
		- Schritt105 => Stop Achse und Übergabe Recording Position an die VAR lr_RecPos


		Konfiguration:
		In der IE Hilfe unter "Funktion Probe Unit" findet man die Beschreibung.
		
		im tsm muss der Touch Probe konfiguriert werden.
		Parameter		Wert		
		S-0-0303		405
		S-0-0307		409
		S-0-0169		1
		S-0-0170		3

		in den Prozessdaten einfügen 
		S-0-0801		Digital inputs, sate			und mit der Var i16_DigitalInput der jeweiligen Achse verknüpfen

		im Drivemanager die Logik der Probe unit einstellen 
		- bei Mux1 den Input auswählen und negiert zuweisen
		- 1: Auto activation from SafeOp to Op auswählen

		PLC:
		im VAR_OUTPUT der Achse die Var anlegen
		lr_RecPos							: LREAL;
		
		im VAR anlegen
		i16_DigitalInput						AT %I* : INT;
	
	
		und im Aufruf fb_axis die Var hinzufügen
	
		lr_RecPos=> lr_RecPos,
		b_TriggerInput:=i16_DigitalInput.2,
		b_FallingEdge:=TRUE


 ========================================================*)
IF	mc_touch_probe.Done THEN
	lr_RecPos:=mc_touch_probe.RecordedPosition;
END_IF


(* Touch Probe Initialisierung *)
TriggerInput.EncoderID:= 	st_masterachse.NcToPlc.AxisId;		(* funktioniert so nur wenn die Encoder ID gleich ist wie die Achs ID*)
TriggerInput.TouchProbe:=	TouchProbe1;					(*bei MC_TouchProbe immer TouchProbe1*)
TriggerInput.Edge:=			RisingEdge;						(*bei MC_TouchProbe immer RisingEdge*)
TriggerInput.Mode:=			TOUCHPROBEMODE_SINGLE;



(* Touch Probe Aufruf *)
mc_touch_probe(
	Execute:= ,
	WindowOnly:= 	FALSE ,
	FirstPosition:= ,
	LastPosition:= ,
	Axis:= 			st_masterachse,
	TriggerInput:=	TriggerInput ,
	Done=> ,
	Busy=> ,
	CommandAborted=> ,
	Error=> ,
	ErrorID=> ,
	RecordedPosition=> );

mc_abort_trigger(
	Execute:= ,
	Axis:= 			st_masterachse,
	TriggerInput:=	TriggerInput ,
	Done=> ,
	Busy=> ,
	Error=> , 
	ErrorID=> );
END_ACTION

(* POU EPT Lib/Funktionsbausteine/ST_CommandHistory, ST *)
FUNCTION_BLOCK ST_CommandHistory
VAR_INPUT
	i16_current_cmd 		: enum_ecd_cmd;
END_VAR
VAR_OUTPUT
	last_cmd 			: enum_ecd_cmd;
END_VAR
VAR
	arr_last_cmd_history 	: ARRAY[0..31] OF enum_ecd_cmd;
	i					: INT;
END_VAR
IF (last_cmd <> i16_current_cmd) THEN
	last_cmd := i16_current_cmd;

	FOR i:= 30 TO 0 BY -1DO
		arr_last_cmd_history[i+1] := arr_last_cmd_history[i];
	END_FOR
	arr_last_cmd_history[0] := last_cmd;
END_IF
END_FUNCTION_BLOCK

(* POU EPT Lib/Achsen/BECKHOFF/ST_AxisJobCtrl_Cam_Gear, ST *)
FUNCTION_BLOCK ST_AxisJobCtrl_Cam_Gear
VAR_INPUT
	r_getriebefaktor						: LREAL;
	r_master_position					: LREAL;
	mc_activation_mode_camin			: MC_CamActivationMode;
	lr_activation_position_camin			: LREAL := 0.0;
	mc_activation_mode_scaleing		: MC_CamActivationMode;
	lr_activation_position_scaleing		: LREAL := 0.0;
	mc_buffermode_axis					: MC_BufferMode;     (*	MC_Aborting,	->sofortiger Abbruch der momentanen Bewegung, bei einem neuen Verfahrbefehl
														MC_Buffered,
														MC_BlendingLow,
														MC_BlendingPrevious,
														MC_BlendingNext,
														MC_BlendingHigh *)
	mc_cam_point_id						: MC_MotionFunctionPoint_ID; (* MC_MotionFunctionPoint_ID : UDINT; *)
	mc_motion_function_point				: MC_MotionFunctionPoint;	(*TYPE MC_MotionFunctionPoint :
																	STRUCT
																	    PointIndex        : MC_MotionFunctionPoint_ID;
																	    FunctionType      : MC_MotionFunctionType;
																	    PointType         : MC_MotionPointType;
																	    RelIndexNextPoint : MC_MotionFunctionPoint_ID;
																	    MasterPos         : LREAL; (* X *)
																	    SlavePos          : LREAL; (* Y *)
																	    SlaveVelo         : LREAL; (* Y' *)
																	    SlaveAcc          : LREAL; (* Y'' *)
																	    SlaveJerk         : LREAL; (* Y''' *)
																	END_STRUCT
																END_TYPE*)
	st_camin_options						: ST_CamInOptions_V2;
	st_camexchange_options				: ST_CamExchangeOptions ;
	mc_cam_table_id					 	: MC_CAM_ID;	(* MC_CAM_ID : UDINT; *)
	mc_reference_cam_table_id				: MC_CAM_ID;	(* MC_CAM_ID : UDINT; *)
	st_camscaling_data						: ST_CamScalingData;	(*STRUCT
																	(* scaling of the X axis of the cam (master scaling) *)
																	MasterScalingMode 	: MC_CamScalingMode;
																	MasterRelative 	: BOOL;
																	MasterOffset 	: LREAL; (* E *)
																	MasterScaling 	: LREAL := 1.0; (* E *)
																
																	(* scaling of the Y axis of the cam (slave scaling) *)
																	SlaveScalingMode 	: MC_CamScalingMode;
																	SlaveRelative 	: BOOL;
																	SlaveOffset 	: LREAL; (* E *)
																	SlaveScaling 	: LREAL := 1.0; (* E *)
																	END_STRUCT*)
END_VAR
VAR_IN_OUT
	st_masterachse						: AXIS_REF;
	st_slaveachse 						: AXIS_REF;
	st_ecd_cmd							: struct_ecd_cmd;
END_VAR
VAR
	fb_ton_cmd_timeout					: TON;
	fb_ton_vz							: TON;
	mc_gearindyn_axis 					: MC_GearInDyn;
	mc_gearout_axis						: MC_GearOut;
	mc_camin_axis						: MC_CamIn_V2;
	mc_camout_axis						: MC_CamOut;
	mc_cam_scaleing						: MC_CamScaling_V2;
	mc_read_motion_function_point			: MC_ReadMotionFunctionPoint;
	mc_write_motion_function_point			: MC_WriteMotionFunctionPoint;
	mc_read_camtable_slave_dynamics		: MC_ReadCamTableSlaveDynamics;
	st_cam_table_characteristics			: MC_TableCharacValues;
	mc_read_camtable_characteristics		: MC_ReadCamTableCharacteristics;
	err_id								: DWORD := 0;
	fb_state_entry							: ST_StateEntry;
	fb_cmd_history						: ST_CommandHistory;
END_VAR
(* Zeiten *)
fb_ton_cmd_timeout(IN:= , PT:= t#5s, Q=> , ET=> );
fb_ton_vz(IN:= , PT:= , Q=> , ET=> );

(* ======================================Schrittkette Drivebefehle======================================== *)
fb_state_entry(
	i16_next_step:= ,
	i16_pos:= 1,
	s_debugtext:= ,
	E=> ,
	X=> ,
	i16_step=> ,
	i16_last_step=> );

